PROC HomeSetup()
 !***********************************************************************
 !* Prozedur zum Programmieren und Parametrieren der Homepositionen 1-5 *
 !*     Procedure for programming and setup the home positions 1-5      *
 !***********************************************************************
 ! Gewaehlte Homeposition / Selected home position
 VAR num n_HomeSelect;
 ! richtigstellen der Homereihenfolge falls erste home deaktiviert / Set default home configuration
 IF b_HomeInUse{1}=FALSE b_HomeInUse:=[TRUE,FALSE,FALSE,FALSE,FALSE];
 WHILE TRUE DO
  TPErase;
  rerun1:
	! Home Liste wird Initialisiert / Create list of homes
  FOR i FROM 1 TO 5 DO
		IF b_HomeInUse{i} THEN
			listHome{i}.text:=listHomeConst{i}.text+st_Home_label{i};
		ELSE
			listHome{i}.text:="";
		ENDIF
  ENDFOR
  !
  ! Waehle Home Nummer
  st_UiHeader:=["Setup Home.","Setup Home, Waehle eine Homepos aus.","???"];
  st_UiMsgButtons3:=["Please select the Home you want to change.","Anzahl der Home aendern","???"];
  st_UiMsgButtons4:=["OK","Ok","???"];
  st_UiMsgButtons5:=["Finished","Beenden","???"];
  st_UiMsgButtons:=["","",st_UiMsgButtons3{n_Sp},st_UiMsgButtons4{n_Sp},st_UiMsgButtons5{n_Sp}];
	n_HomeSelect := UIListView(\Result:=br_UiAnswer\Header:=st_UiHeader{n_Sp},listHome
 	  \BtnArray:=st_UiMsgButtons\Icon:=iconInfo\DefaultIndex:=1);
  IF br_UiAnswer = 5 THEN
  	TPErase;
  	TPShow TP_LATEST;
    RETURN;
  ENDIF
  IF br_UiAnswer = 3 THEN
		! Anzahl der verwendeten Homes\Number of used homes
		st_UiHeader:=["Enter number of homes used","Anzahl der verwendeten Home Positonen","???"];
		st_UiMsgLine1:=["   count 1-5","   Anzahl 1-5","???"];
		n_Temp := UINumEntry(\Header:=st_UiHeader{n_Sp}\Message:=st_UiMsgLine1{n_Sp}\Icon:=iconInfo
			\InitValue:=1\MinValue:=1\MaxValue:=5\AsInteger);
		!
		TEST n_Temp
			CASE 1:
				b_HomeInUse:=[TRUE,FALSE,FALSE,FALSE,FALSE];
				b_HomeAkt:=[TRUE,FALSE,FALSE,FALSE,FALSE];
			CASE 2:
				b_HomeInUse:=[TRUE,TRUE,FALSE,FALSE,FALSE];
				b_HomeAkt:=[TRUE,TRUE,FALSE,FALSE,FALSE];
			CASE 3:
				b_HomeInUse:=[TRUE,TRUE,TRUE,FALSE,FALSE];
				b_HomeAkt:=[TRUE,TRUE,TRUE,FALSE,FALSE];
			CASE 4:
				b_HomeInUse:=[TRUE,TRUE,TRUE,TRUE,FALSE];
				b_HomeAkt:=[TRUE,TRUE,TRUE,TRUE,FALSE];
      CASE 5:
      	b_HomeInUse:=[TRUE,TRUE,TRUE,TRUE,TRUE];
      	b_HomeAkt:=[TRUE,TRUE,TRUE,TRUE,TRUE];
     ENDTEST
     GOTO rerun1;
	ENDIF
  !
  rerun2:
  ! was soll geaendert werden / what should be changed
  n_Temp :=0;
  st_UiHeader:=["Setup homepos edit Home_","Setup Home, bearbeite Home_","???"];
  st_UiMsgLine1:=["Modify the position Home_","aendere die Position der Home_","???"];
  st_UiMsgLine2:=["Modify the description for Home_","aendere die Beschreibung fuer die Home_","???"];
  st_UiMsgLine3:=["Activate the output for Home_","Aktiviere den Ausgang fuer die Home_","???"];
  st_UiMsgButtons3:=["Return","Zurueck","???"];
  st_UiMsgButtons4:=["OK","OK","???"];
  st_UiMsgButtons5:=["Finished","Beenden","???"];
  st_UiMsgButtons:=["","",st_UiMsgButtons3{n_Sp},st_UiMsgButtons4{n_Sp},st_UiMsgButtons5{n_Sp}];
  li_UiMsgList:=[["",st_UiMsgLine1{n_Sp}+NumToStr(n_HomeSelect,0)],["",st_UiMsgLine2{n_Sp}+NumToStr(n_HomeSelect,0)]
  	,["",st_UiMsgLine3{n_Sp}+NumToStr(n_HomeSelect,0)],["",""],["",""]];
  n_Temp := UIListView(\Result:=br_UiAnswer\Header:=st_UiHeader{n_Sp}+NumToStr(n_HomeSelect,0),li_UiMsgList
  		\BtnArray:=st_UiMsgButtons\Icon:=iconInfo\DefaultIndex:=1);
	IF br_UiAnswer = 5 THEN
		TPErase;
		TPShow TP_LATEST;
		RETURN;
	ENDIF
	! zurueck zur auswahl / back to selection
	IF br_UiAnswer=3 GOTO rerun1;
	! auswahl aendere Pos / Select home to change
	IF n_Temp=1 THEN
		br_UiAnswer:=0;
		st_UiHeader:=["Setup homepos edit Home_","Setup Home, neue Pos fuer Home_","???"];
		st_UiMsgLine1:=["Make the current Position the new Home_"+NumToStr(n_HomeSelect,0)+" positon!","Die aktuell Position wird als Home_"+NumToStr(n_HomeSelect,0)+" gespeichert!","???"];
		st_UiMsgButtons3:=["Return","Zurueck","???"];
		st_UiMsgButtons4:=["   Save    Position?","Position speichern!","???"];
		st_UiMsgButtons5:=["Finished","Beenden","???"];
		st_UiMsgButtons:=["","",st_UiMsgButtons3{n_Sp},st_UiMsgButtons4{n_Sp},st_UiMsgButtons5{n_Sp}];
		br_UiAnswer:= UIMessageBox (\Header:=st_UiHeader{n_Sp}+NumToStr(n_HomeSelect,0)
			\Message:=st_UiMsgLine1{n_Sp}\BtnArray:=st_UiMsgButtons\Icon:=iconWarning);
		IF br_UiAnswer = 5 THEN
			TPErase;
			TPShow TP_LATEST;
			RETURN;
		ENDIF
		! Pos fuer die jeweilige Home zuweisen / Pos assign for each Home
		IF br_UiAnswer = 4 THEN
			t_Home := CTool();
			t_home.robhold:=TRUE;
		TEST n_HomeSelect
			CASE 1:
				jpHome1 := CJointT();
				robjOHome1:=jpHome1.robax;
				extjOHome1:=jpHome1.extax;
			CASE 2:
				jpHome2 := CJointT();
				robjOHome2:=jpHome2.robax;
				extjOHome2:=jpHome2.extax;
			CASE 3:
				jpHome3 := CJointT();
				robjOHome3:=jpHome3.robax;
				extjOHome3:=jpHome3.extax;
			CASE 4:
				jpHome4 := CJointT();
				robjOHome4:=jpHome4.robax;
				extjOHome4:=jpHome4.extax;
			CASE 5:
				jpHome5 := CJointT();
				robjOHome5:=jpHome5.robax;
				extjOHome5:=jpHome5.extax;
			ENDTEST
			! ungueltig setzen / error set
			b_HomeAkt{n_HomeSelect}:=FALSE;
		GOTO rerun2;
	ENDIF
 ENDIF
 ! ruecksprung ins aenderungsmenue / jump back into the change of menu
 IF br_UiAnswer = 3 GOTO rerun2;
 ! auswahl aendere beschreibung / selection change description
 IF n_Temp=2 THEN
 	st_UiHeader:=["Setup homepos edit Home_","Setup Home, Beschreibung fuer Home_","???"];
	st_UiMsgLine1:=["Please enter the new description","Bitte eine Beschreibung fuer die HomePos eingeben.","???"];
	st_Home_label{n_HomeSelect} := UIAlphaEntry(\Header:=st_UiHeader{n_Sp}+NumToStr(n_HomeSelect,0),
	  \Message:=st_UiMsgLine1{n_Sp}\Icon:=iconInfo\InitString:= st_Home_label{n_HomeSelect});
	GOTO rerun2;
 ENDIF
 ! auswahl aktiviere Ausgang / Output enable selection
 IF n_Temp=3 THEN
	br_UiAnswer:=0;
	st_UiHeader:=["Setup homepos edit Home_","Setup Home, Ausgang fuer Home_","???"];
	st_UiMsgLine1:=["In order to activate the Home output, you must Warm Start the controller.","Der Ausgang fuer die Home wird durch einen Warmstart aktiviert!","???"];
	st_UiMsgButtons1:=["Warmstart!","Warmstart!","???"];
	st_UiMsgButtons3:=["Return","Zurueck","???"];
	st_UiMsgButtons5:=["Finished","Beenden","???"];
	st_UiMsgButtons:=[st_UiMsgButtons1{n_Sp},"",st_UiMsgButtons3{n_Sp},"",st_UiMsgButtons5{n_Sp}];
	br_UiAnswer:= UIMessageBox (\Header:=st_UiHeader{n_Sp}+NumToStr(n_HomeSelect,0)
	\Message:=st_UiMsgLine1{n_Sp}\BtnArray:=st_UiMsgButtons\Icon:=iconWarning);
	IF br_UiAnswer = 5 THEN
		TPErase;
		TPShow TP_LATEST;
		RETURN;
		ENDIF
		IF br_UiAnswer = 3 GOTO rerun2;
		IF br_UiAnswer = 1 WarmStart;
	ENDIF
 ENDWHILE
ENDPROC !(HomeSetup)

!*******************************************************************************

PROC SyncPosSetup()
 !******************************
 !*     Sync Switch Setup      *
 !******************************
 br_UiAnswer:=0;
 st_UiHeader:=["Setup SyncPos","Setup Synchron Position","???"];
 st_UiMsgLine1:=["Please note only use when the robot is at the ","Achtung  nur wenn der Roboter den Synchronschalter belegt","???"];
 st_UiMsgLine2:=["synchronous switch or on the soft-synchronous ","oder auf der Soft-Synchronposition steht","???"];
 st_UiMsgLine3:=["position. Otherwise, press> 'Abort'!","diese Position speichern. Ansonsten den Vorgang abbrechen!","???"];
 st_UiMsgButtons4:=["Save Position!","Position speichern!","???"];
 st_UiMsgButtons5:=["Abort","Abbruch","???"];
 st_UiMsgButtons:=["","","",st_UiMsgButtons4{n_Sp},st_UiMsgButtons5{n_Sp}];
 st_UiMsgLines:=[st_UiMsgLine1{n_Sp},st_UiMsgLine2{n_Sp},st_UiMsgLine3{n_Sp},"",""];
 br_UiAnswer:= UIMessageBox (\Header:=st_UiHeader{n_Sp}
		\MsgArray:=st_UiMsgLines\BtnArray:=st_UiMsgButtons\Icon:=iconWarning);
 IF br_UiAnswer = 5 THEN
	TPErase;
	TPShow TP_LATEST;
	RETURN;
 ENDIF
 ! Pos zuweisen
 IF br_UiAnswer = 4 THEN
	t_SMSync := CTool();
	t_SMSync.robhold:=TRUE;
	jpSM1SyncSwitch := CJointT(\TaskRef:=T_ROB1Id);
	robjOSM1SyncSwitch:=jpSM1SyncSwitch.robax;
	extjOSM1SyncSwitch:=jpSM1SyncSwitch.extax;
 ENDIF
 TPErase;
 TPShow TP_LATEST;
ENDPROC !(SynchPosSetup)

!*******************************************************************************

FUNC num n_RobInHomeDO()
 !*****************************************************************************************
 !* Funktion Ueberprueft die Home Ausgaenge des Roboters und gibt entsprechend 1-5 zurueck *
 !*        Function to return the number in which home the robot is at (1-5)              *
 !*****************************************************************************************
 !
 IF DOutput(SYS_do_Home_1)=1 THEN
   RETURN 1;
 ELSEIF DOutput(SYS_do_Home_2)=1 THEN
   RETURN 2;
 ELSEIF DOutput(SYS_do_Home_3)=1 THEN
   RETURN 3;
 ELSEIF DOutput(SYS_do_Home_4)=1 THEN
   RETURN 4;
 ELSEIF DOutput(SYS_do_Home_5)=1 THEN
   RETURN 5;
 ELSE
   RETURN 0;
 ENDIF
ENDFUNC !(n_RobInHomeDO)

!*******************************************************************************

FUNC bool b_PLCNeedHome(num n_H)
 !***********************************************************
 !* Function to check which home the PLC requires the robot *
 !***********************************************************
 !
 TEST n_H
 	CASE 1:
		IF DInput(PLC_di_Home_1)=1 RETURN TRUE;
 		RETURN FALSE;
  CASE 2:
 		IF DInput(PLC_di_Home_2)=1 RETURN TRUE;
  	RETURN FALSE;
  CASE 3:
  	IF DInput(PLC_di_Home_3)=1 RETURN TRUE;
  	RETURN FALSE;
  CASE 4:
  	IF DInput(PLC_di_Home_4)=1 RETURN TRUE;
  	RETURN FALSE;
  CASE 5:
  	IF DInput(PLC_di_Home_5)=1 RETURN TRUE;
  	RETURN FALSE;
  DEFAULT :
    	RETURN FALSE;
 ENDTEST
ENDFUNC !(b_PLCNeedHome)

!*******************************************************************************

PROC CheckValue(num Value,num MinValue,num MaxValue,num Dec,string Header)
 !**************************************************************************************************
 !*            Prozedur Ueberprueft ob ein Wert innerhalb eines Bereiches liegt                    *
 !* uebergebene Parameter: num Value,num MinValue,num MaxValue,num Dec,string Header (fuer meldung) *
 !*                         Check values are within certain paramaters                             *
 !**************************************************************************************************
 WHILE Value<MinValue OR Value>MaxValue DO
  st_UiHeader:=["Value Error ","Falscher Wert von ","???"];
  st_UiMsgLine1:=["The value is outside the Min or Max range.","Wert ist ausserhalb des gueltigen Bereichs","???"];
  st_UiMsgLine2:=["Min Value= ","Minnimal Wert= ","???"];
  st_UiMsgLine3:=["Max Value= ","Maximal  Wert= ","???"];
  st_UiMsgLine4:=["The Programmed Value=","Programmierter Wert= ","???"];
  UIMsgBox\Header:=st_UiHeader{n_Sp}+Header, st_UiMsgLine1{n_Sp}\MsgLine2:=st_UiMsgLine2{n_Sp}+NumToStr(MinValue,Dec)
 		 \MsgLine3:=st_UiMsgLine3{n_Sp}+NumToStr(MaxValue,Dec) \MsgLine4:=st_UiMsgLine4{n_Sp}+NumToStr(Value,Dec)
  		\Buttons:=btnOK\Icon:=iconWarning;
	Stop ;
	ENDWHILE
ENDPROC !(CheckValue)

!*******************************************************************************

PROC PowerOnCom()
 !***************************************************
 !* Abfrage der Appl im System nach einem Warmstart *
 !*        Check system after a warm start          *
 !***************************************************
 !Appl-Feld wird geloescht / Applications-deleted box
 VAR bool b_ComDummy:=FALSE;
 VAR bool b_timeout;
 VAR num n_ComDummy:=0;
 VAR NUM n_error_offset_x:=0 ;
 VAR NUM n_error_offset_y:=0 ;
 VAR NUM n_error_offset_z:=0 ;
 VAR bool b_ABS_Acc_Enable_MEM:=TRUE;
 VAR string st_CFG_RobotType;

 b_PwOnEnd:=FALSE;
 Reset VB_do_TaskBrake;
 FOR I FROM 1 TO 30 DO
	b_Start_present{I}:=TRUE;
	b_ReStart_present{I}:=TRUE;
	b_Stop_present{I}:=TRUE;
	b_Reset_present{I}:=TRUE;
 ENDFOR
 b_StartUser_present:=TRUE;
 b_ReStartUser_present:=TRUE;
 b_StopUser_present:=TRUE;
 b_ResetUser_present:=TRUE;
 ! Appl Info loeschen
 n_ApplMax:=0;
 n_Fk4ApplAktiv:=0;
 b_ABS_Acc_Enable:=TRUE;

 !Abfrage der einzelnen Appls / Check individual Applications
 n_ComDummy:=0;
 FOR I FROM 1 TO 30 DO
  b_ComDummy:=TRUE;
  st_Appl_Info{I,1}:="";
  st_Appl_Info{I,2}:="";
  st_Appl_Info{I,3}:="";
  ! aufruf der PowerOn jeder Appl und einlesen der Strings / calling the PowerOn Appl and read each of the strings
  n_Fk4ApplNum:=I;
  %"PowerON"+NumToStr(I,0)%;
  !
  IF b_ComDummy=TRUE THEN
    Incr n_ComDummy;
    st_Appl_Info{n_ComDummy,1}:=ValToStr(I);
    st_Appl_Info{n_ComDummy,2}:=st_Appl_Name;
    st_Appl_Info{n_ComDummy,3}:=st_Appl_Key{n_Sp};
 	  Incr n_ApplMax;
  ENDIF
 ENDFOR
 n_Fk4ApplNum:=0;

b_TbCom_Started:=FALSE ;

Waituntil b_TbCom_Started=TRUE\MaxTime:= 50\TimeFlag:= b_timeout;
!***************************
!* Waiting TB_Com to start *
!***************************

 b_PowerOn_exe_OK:=TRUE ;

 ! setzen der Homepos als Weltzonen / share of the world as Homepos Zones
 !
 IF b_HomeInUse{1}=TRUE THEN
    WZHomeJointDef \Inside, sh_HomePos1, jpHome1, delta_HomePosFine;
    WZDOSet \Stat,wz_HomePos1 \Inside, sh_HomePos1, SYS_do_Home_1,high;
    b_HomeAkt{1}:=TRUE;
 ENDIF
 !
 IF b_HomeInUse{2}=TRUE THEN
     WZHomeJointDef \Inside, sh_HomePos2, jpHome2, delta_HomePosFine;
     WZDOSet \Stat,wz_HomePos2 \Inside, sh_HomePos2, SYS_do_Home_2,high;
     b_HomeAkt{2}:=TRUE;
 ENDIF
 !
 IF b_HomeInUse{3}=TRUE THEN
     WZHomeJointDef \Inside, sh_HomePos3, jpHome3, delta_HomePosFine;
     WZDOSet \Stat,wz_HomePos3 \Inside, sh_HomePos3, SYS_do_Home_3,high;
     b_HomeAkt{3}:=TRUE;
 ENDIF
 !
 IF b_HomeInUse{4}=TRUE THEN
     WZHomeJointDef \Inside, sh_HomePos4, jpHome4, delta_HomePosFine;
     WZDOSet \Stat,wz_HomePos4 \Inside, sh_HomePos4, SYS_do_Home_4,high;
     b_HomeAkt{4}:=TRUE;
 ENDIF
 !
 IF b_HomeInUse{5}=TRUE THEN
     WZHomeJointDef \Inside, sh_HomePos5, jpHome5, delta_HomePosFine;
     WZDOSet \Stat,wz_HomePos5 \Inside, sh_HomePos5, SYS_do_Home_5,high;
     b_HomeAkt{5}:=TRUE;
 ENDIF
 !
 ! Poweron fuer Anwender wenn noetig / Poweron for users if necessary
 %"PowerOnUser"%;
 !---------------
 ! Copy SM_Files and Backup files
 SM1_CopyCfg;
 CopyCfg;

b_PwOnEnd:=TRUE;
b_ABS_Acc_Enable_MEM:=b_ABS_Acc_Enable;

 !Get robot type
 ReadCfgData "/MOC/ROBOT/ROB_1","use_robot_type",st_CFG_RobotType;

 st_RobotType:=st_CFG_RobotType;

 !Set Absoulute accuracy flag
 TEST st_RobotType

 CASE "ROB1_6620LX_1.90_150":
 	b_Robot_ABS_Type:=FALSE;
 DEFAULT:
 	b_Robot_ABS_Type:=b_ABS_Acc_Enable_MEM;
 ENDTEST

 !Set output as this robot does not use this output
 IF st_RobotType="ROB1_6620LX_1.90_150" Set SM1_do_Stopped;

 IF b_Robot_ABS_Type THEN
	! Abfrage ob die AbsAcc ein ist
	ReadCfgData "/MOC/ROBOT/ROB_1","use_robot_calib",st_Abs;

	IF st_Abs="r1_uncalib" THEN
		st_UiHeader:=["Com, Absolute Accuracy error","Com, Keine Absolutgenauigkeit","???"];
		st_UiMsgLine1:=["Warning!! The robot absolute accuracy is turned Off.","Ohne Absolutgenauigkeit ist es nicht erlaubt den Roboter ","???"];
		st_UiMsgLine2:=["There is a risk of collisions!","zu bewegen, es besteht Kollisionsgefahr!","???"];
		st_UiMsgLine3:=["Please ensure it is enabled!","Bitte schalten Sie die Absolutgenauigkeit wieder ein!","???"];
		ErrWrite st_UiHeader{n_Sp},st_UiMsgLine1{n_Sp} \RL2:=st_UiMsgLine2{n_Sp}\RL3:=st_UiMsgLine3{n_Sp};
	ELSE
		!Check absolute accurate data exist
		ReadCfgData "/MOC/ARM_CALIB/rob1_1", "error_offset_x", n_error_offset_x;
		ReadCfgData "/MOC/ARM_CALIB/Rob1_1", "error_offset_y", n_error_offset_y;
		ReadCfgData "/MOC/ARM_CALIB/Rob1_1","error_offset_z",n_error_offset_z;

		IF n_error_offset_x=0 AND n_error_offset_y=0 AND n_error_offset_z=0 THEN
			st_UiHeader:=["Com, Absolute Accuracy error","Com, Keine Absolutgenauigkeit","???"];
			st_UiMsgLine1:=["Warning!! The robot absolute accuracy is turned On but,","Warnung!! Der Roboter absolute Genauigkeit ist eingeschaltet,","???"];
			st_UiMsgLine2:=["the 'ARM/JOINT_CALIB' data in the 'MOC.cfg' file","aber die 'ARM/JOINT_CALIB' Daten in der 'MOC.cfg'","???"];
			st_UiMsgLine3:=["may not exist.","Datei kann nicht vorhanden","???"];
			st_UiMsgLine4:=["Please check.","Bitte überprüfen.","???"];

			ErrWrite st_UiHeader{n_sp},st_UiMsgLine1{n_sp} \RL2:=st_UiMsgLine2{n_sp}\RL3:=st_UiMsgLine3{n_sp}\RL4:=st_UiMsgLine4{n_sp};
		ENDIF
	ENDIF
 ENDIF

 ERROR
 !** Error Handler**
 SkipWarn;

 TEST ERRNO
 CASE ERR_CFG_NOTFND:
   TRYNEXT;

 CASE ERR_REFUNKPRC:
   b_ComDummy:=FALSE;
   st_Appl_Name:="";
   st_Appl_Key:=["","",""];
   TRYNEXT;
 ENDTEST
ENDPROC !(PowerOnCom)

!*******************************************************************************

PROC StartCom()
 !****************************
 !* Aufruf der Startroutinen *
 !*     Start Routine        *
 !****************************
 VAR bool b_ComDummy:=FALSE;
 VAR num n_ComDummy:=0;
 ! ob Programmzeiger versetzt wurde / whether program pointer was moved
 IF PPMovedInManMode() ResetPPMoved;
 !
 IF b_CheckPP=FALSE THEN
	Reset SYS_do_MainStarted;
	! loeschen von Fehlern wenn neustart / Clear errors after new start
	SetGO PLC_go_ErrCode, 0;
	Reset PLC_do_MsgToPLC;
	Reset PLC_do_ErrorToPLC;
	Reset PLC_do_StopToPLC;
	MsgBox_Clear;
	b_CollClearAct:= FALSE;
	n_JobReqNum:=0;
	n_JobFinNum:=0;
	b_JobF_w:=FALSE;
	b_JobR_w:=FALSE;
 ENDIF

 ! aufruf der Eventroutinen der Appl / calling the routines in the events
 b_UserEv:=FALSE;
 IF n_ApplMax >0 AND n_ApplMax< 31 THEN
	FOR I FROM 1 TO n_ApplMax DO
		n_Appl_count:=I;
		IF (st_Appl_Info{I,1}="") OR (b_Start_present{I}=FALSE) GOTO END_Start;
		b_ComDummy:=StrToVal(st_Appl_Info{I,1},n_ComDummy);
		%"Start"+NumToStr(n_ComDummy,0)%;
	 	END_Start:
	ENDFOR
 ENDIF

 IF n_ModeOP_Mem<>OpMode() THEN
      b_Ignore_NoAppl_Chk:=FALSE ;
      n_ModeOP_Mem:=OpMode();
 ENDIF

 IF PLC_di_NoApplication=1 AND b_Ignore_NoAppl_Chk=FALSE THEN
    MsgBoxEv_Clear;
    st_MsgBoxEvHeader:=["Warning!! StartCom","Warnung!! StartCom","???"];
	st_Dummy:=["You are about to run with (PLC_di_NoApplication=1)","Du bist zum Laufen (PLC_di_NoApplication=1)","???"];
	st_MsgBoxEvLine3:=["no Application selected.","nein Anwendung ausgewaehlt.","???"];
    st_MsgBoxEvbutton4:=["Continue","OK","???"];

	IF OpMode()<>OP_Auto THEN
		st_MsgBoxEvLine5:=["Press>'Ignore' to stop message re-occuring.","Druecke> 'Ignorieren' um die Nachricht zu stoppen.","???"];
		st_MsgBoxEvbutton5:=["Ignore","Ignorieren","???"];
   ENDIF

    MsgBoxEv\line1:=""\Line2:=st_Dummy{n_Sp};

    IF n_MsgBoxEvAnswer=5 b_Ignore_NoAppl_Chk:=TRUE;
 ENDIF

 b_UserEv:=TRUE;
 IF b_StartUser_present = TRUE %"StartUser"%;
 !
 ERROR
 !** Error Handler**
 IF ERRNO=ERR_REFUNKPRC THEN
 	SkipWarn;
	IF b_UserEv=TRUE THEN
		b_StartUser_present:=FALSE;
	ELSE
		b_Start_present{n_Appl_count}:=FALSE;
 	ENDIF
	TRYNEXT;
 ENDIF
ENDPROC !(StartCom)

!*******************************************************************************

PROC StopCom()
 !***************************
 !* Aufruf der Stoproutinen *
 !*     Stop Routine        *
 !***************************
 VAR bool b_ComDummy:=FALSE;
 VAR num n_ComDummy:=0;
 ! ob Programmzeiger versetzt wurde / whether program pointer was moved
 IF b_CheckPP=FALSE   Reset SYS_do_MainStarted;
 ! aufruf der Eventroutinen der Appl / calling the routines in the events
 b_UserEv:=FALSE;
 IF n_ApplMax >0 AND n_ApplMax< 31 THEN
	FOR I FROM 1 TO n_ApplMax DO
		n_Appl_count:=I;
		IF (st_Appl_Info{I,1}="") OR (b_Stop_present{I}=FALSE) GOTO END_Stop;
		b_ComDummy:=StrToVal(st_Appl_Info{I,1},n_ComDummy);
		%"Stop"+NumToStr(n_ComDummy,0)%;
	 	END_Stop:
	 ENDFOR
 ENDIF
 b_UserEv:=TRUE;
 IF b_StopUser_present = TRUE %"StopUser"%;
 ERROR
 !** Error Handler**
 IF ERRNO=ERR_REFUNKPRC THEN
 	SkipWarn;
	IF b_UserEv=TRUE THEN
		b_StopUser_present:=FALSE;
	ELSE
		b_Stop_present{n_Appl_count}:=FALSE;
 	ENDIF
	TRYNEXT;
 ENDIF
ENDPROC !(StopCom)

!*******************************************************************************

PROC RestartCom()
 !******************************
 !* Aufruf der ReStartroutinen *
 !*     Re-Start Routine       *
 !******************************
 VAR bool b_ComDummy:=FALSE;
 VAR num n_ComDummy:=0;
 VAR errnum errno1;
 ! ob Programmzeiger versetzt wurde / whether program pointer was moved
 b_PPMoved:=FALSE;
 IF PPMovedInManMode() THEN
	b_PPMoved:=TRUE;
	! loeschen von Fehlern wenn start / Clear errors if Restart
	SetGO PLC_go_ErrCode, 0;
	Reset PLC_do_MsgToPLC;
	Reset PLC_do_ErrorToPLC;
	Reset PLC_do_StopToPLC;
	MsgBox_Clear;
	MsgBoxEv_Clear;
	b_CollClearAct:= FALSE;
	b_JobF_w:=FALSE;
	b_JobR_w:=FALSE;

     IF DOutput(SYS_do_MainStarted)=1 AND DOutput (SYS_do_ApplRun)=1 AND b_PPMoved_mem=FALSE THEN
         b_PPMoved_mem:=TRUE;
         Log_Message "STD","Program pointer moved in Manual mode";
     ENDIF

 ENDIF

 IF OpMode()=OP_AUTO b_PPMoved_mem:=FALSE;

 IF b_CheckPP=FALSE   Reset SYS_do_MainStarted;
 ! aufruf der Eventroutinen der Appl / calling the routines in the events
 b_UserEv:=FALSE;
 IF n_ApplMax >0 AND n_ApplMax< 31 THEN
		FOR I FROM 1 TO n_ApplMax DO
			n_Appl_count:=I;
			IF (st_Appl_Info{I,1}="") OR (b_ReStart_present{I}=FALSE)  GOTO END_Restart;
			b_ComDummy:=StrToVal(st_Appl_Info{I,1},n_ComDummy);
			%"Restart"+NumToStr(n_ComDummy,0)%;
			END_Restart:
		ENDFOR
	ENDIF

 b_UserEv:=TRUE;
 IF b_ReStartUser_present = TRUE %"RestartUser"%;
 ! abfrage auf simulierte signale
 IF DOutput(VB_do_Simulated_IO)= 1 AND OpMode()= OP_AUTO  AND RobOs() = TRUE THEN
	! Meldung an SPS
	SetGO PLC_go_ErrCode, 34;
	Set PLC_do_MsgToPLC;
 	WHILE DOutput(VB_do_Simulated_IO)= 1 AND OpMode()= OP_AUTO DO
  		st_UiHeader:=["Com, Caution simulated signals!","Com, Achtung Simulierte Signale!","???"];
  		st_UiMsgLine1:=["There are some signals that are simulated which is not allowed in","Das Simulieren von Signalen ist im Automatik nicht erlaubt!","???"];
  		st_UiMsgLine2:=["automatic mode!  Please switch to manual mode,","In die Betriebsart Hand wechseln und die","???"];
  		st_UiMsgLine3:=["select the I/O menu then turn off the simulation/s.","Simulation aller Signale im Ein-Ausgangs Fenster ausschalten.","???"];
  		UIMsgBox\Header:=st_UiHeader{n_Sp},st_UiMsgLine1{n_Sp}\MsgLine2:=st_UiMsgLine2{n_Sp}\MsgLine3:=st_UiMsgLine3{n_Sp}
  						\Buttons:=btnNone\Icon:=iconError\MaxTime:=1.5\BreakFlag:=errno1;
			!
	ENDWHILE
 	SetGO PLC_go_ErrCode, 0;
 	Reset PLC_do_MsgToPLC;
 ENDIF
 ! check SafeMove function,at error to reduce speed
 IF DOutput(SM1_do_BrakeReq) =0 THEN
  	VelSet 100,5000;
 ELSE
  	VelSet 100,150;
		ErrWrite \W, "ComBase, SM1_do_BrakeReq =1", "Speed reduce to 150mm/s" ;
 ENDIF

 IF n_ModeOP_Mem<>OpMode() THEN
      b_Ignore_NoAppl_Chk:=FALSE ;
      n_ModeOP_Mem:=OpMode();
 ENDIF

ResetPPMoved;

 ERROR
 !** Error Handler**
 IF ERRNO=ERR_REFUNKPRC THEN
 	SkipWarn;
	IF b_UserEv=TRUE THEN
		b_ReStartUser_present:=FALSE;
	ELSE
		b_ReStart_present{n_Appl_count}:=FALSE;
 	ENDIF
	TRYNEXT;
 ENDIF
ENDPROC !(RestartCom)

!*******************************************************************************

PROC ResetCom()
 !****************************
 !* Aufruf der Resetroutinen *
 !*      Reset Routine       *
 !****************************
 VAR bool b_ComDummy:=FALSE;
 VAR num n_ComDummy:=0;
 ! aufruf der Eventroutinen der Appl / calling the routines in the events
 b_UserEv:=FALSE;
 IF n_ApplMax >0 AND n_ApplMax< 31 THEN
	FOR I FROM 1 TO n_ApplMax DO
		n_Appl_count:=I;
		IF (st_Appl_Info{I,1}="") OR (b_Reset_present{I}=FALSE) GOTO END_Reset;
		b_ComDummy:=StrToVal(st_Appl_Info{I,1},n_ComDummy);
		%"Reset"+NumToStr(n_ComDummy,0)%;
	 	END_Reset:
	ENDFOR
 ENDIF
 b_UserEv:=TRUE;
 IF b_ResetUser_present = TRUE %"ResetUser"%;
 ERROR
 !** Error Handler**
 IF ERRNO=ERR_REFUNKPRC THEN
 	SkipWarn;
	IF b_UserEv=TRUE THEN
		b_ResetUser_present:=FALSE;
	ELSE
		b_Reset_present{n_Appl_count}:=FALSE;
 	ENDIF
	TRYNEXT;
 ENDIF
ENDPROC !(ResetCom)

!*******************************************************************************

FUNC bool b_RobInHomeDO(num Home)
 !************************************************************************************
 !*                            Funktion b_RobInHomeDO                                *
 !* Funktion Ueberprueft die Home Ausgaenge des Roboters und gibt FALSE/TRUE zurueck *
 !*     Function checks the robot exits the home and gives FALSE / TRUE back         *
 !************************************************************************************
  IF Home = 1 AND DOutput(SYS_do_Home_1)=1 THEN
    RETURN TRUE;
  ELSEIF Home = 2 AND DOutput(SYS_do_Home_2)=1 THEN
    RETURN TRUE;
  ELSEIF Home = 3 AND DOutput(SYS_do_Home_3)=1 THEN
    RETURN TRUE;
  ELSEIF Home = 4 AND DOutput(SYS_do_Home_4)=1 THEN
    RETURN TRUE;
  ELSEIF Home = 5 AND DOutput(SYS_do_Home_5)=1 THEN
    RETURN TRUE;
  ELSE
    RETURN FALSE;
  ENDIF
ENDFUNC !(b_RobInHomeDO)

!*******************************************************************************

PROC SM1_CopyCfg()
 !**********************************************
 !* Routine to copy savemove config cfg files  *
 !**********************************************

 VAR string stSMCalFileInt;
 VAR string stSMFileInt;
 VAR string stSMCalFileHome;
 VAR string stSMFileHome;
 VAR string stSMCalFileBck;
 VAR string stSMFileBck;
 VAR string stBckName;
 VAR num n_index;
 ! create folder
 MakeDir "HOME:/SafetyBCK";
 FOR i FROM 1 TO 4 DO
 	! Check all files
	stSMCalFileHome:= stSMCalHome+ ValToStr(i)+ ".xml";
  stSMCalFileInt:= stSMCalInternal+ ValToStr(i)+ ".xml";
  stSMFileHome:= stSMHome+ ValToStr(i)+ ".sxml";
  stSMFileInt:= stSMInternal+ ValToStr(i)+ ".sxml";
  ! If file has a config then safe to Home
	IF FileSize(stSMFileInt) > nSMFilesize THEN
	  	IF IsFile(stSMFileHome) THEN
	   		! delete existing file at Homefolder
	  		RemoveFile stSMFileHome;
	 	  ENDIF
	    IF IsFile(stSMCalFileHome) THEN
	   		! delete existing file at Homefolder
	  		RemoveFile stSMCalFileHome;
	    ENDIF
	    ! Copy actual config from System
	 		CopyFile stSMFileInt, stSMFileHome;
	 		CopyFile stSMCalFileInt, stSMCalFileHome;
			! Read Pin code
			WaitTime 0.2;
			IF IsFile(stSMFileHome) n_SMPins{i}:= GetPinCode(stSMFileHome);
	 ELSE
	 		! Read Backup name
			n_index:=0;
			ReadCfgData "/MMC/BACKUP_DEFAULT/backup_path//hd0a/BACKUP","backup_name",stBckName\ListNo:=n_index;
			stSMFileBck:= stSMBck+ stBckName+ stSMBckFile+ ValToStr(i)+ ".sxml";
			stSMCalFileBck:= stSMBck+ stBckName+ stSMBckCal+ ValToStr(i)+ ".xml";
			! Check on exist config at Backupfolder and right Pin
			! it is for restoring SafeMove config
			IF  IsFile(stSMFileBck)THEN
				 IF (n_SMPins{i} = GetPinCode(stSMFileBck)) THEN
		  			! delete existing file and Copy actual config to System
			  		RemoveFile stSMFileInt;
	  				CopyFile stSMFileBck, stSMFileInt;
		  			ErrWrite \I, "Com, PowerON", "SafeMove, Configfile re-established";
			  		IF  IsFile(stSMCalFileBck)THEN
			  			RemoveFile stSMCalFileInt;
				  		CopyFile stSMCalFileBck, stSMCalFileInt;
					  	ErrWrite \I, "Com, PowerON", "SafeMove, Calfile re-established";
					  ENDIF
			 	 ENDIF
			ENDIF
		ENDIF
 ENDFOR
 !
 ERROR
 !** Error Handler**
 IF ERRNO = ERR_FILEEXIST THEN
  	SkipWarn;
	!Do Nothing
 ELSEIF ERRNO = ERR_FILEACC THEN
  	SkipWarn;
	TRYNEXT;
 ENDIF
 IF ERRNO = ERR_CFG_NOTFND THEN
 	ErrWrite "ComBase /PowerOn", "Path to save SM-Data not correct!" \RL2:="Change the Path in SM1_CopyCfg";
 ENDIF
ENDPROC !(SM1_CopyCfg)

!*******************************************************************************

PROC CopyCfg()
 !************************************************
 !* Routine to copy config cfg files for backup  *
 !************************************************

 VAR string stBckName;
 VAR num n_index;

 ! create folder
 MakeDir "HOME:";

 !Get Backuip name
 ReadCfgData "/MMC/BACKUP_DEFAULT/backup_path//hd0a/BACKUP","backup_name",stBckName\ListNo:=n_index;

 !Create backup Directory name
  IF RobOS() THEN
     stCon_Int_Dir:="/hd0a/internal";
     stCon_Home_Dir:="/hd0a/"+stBckName+"/Home";
     sthd0a_Home_Dir:="/hd0a/Backup/"+stBckName+"/Home";
 ELSE
    stCon_Int_Dir:="INTERNAL:";
    stCon_Home_Dir:="HOME:";
    sthd0a_Home_Dir:="HOME:";
 ENDIF

 !Copy IPaddress file to internal home directory
 IF IsFile(stCon_Int_Dir + "/mc.cfg") THEN

   !Delete old file
    IF IsFile(stCon_Home_Dir + "/mc.cfg") RemoveFile stCon_Home_Dir + "/mc.cfg";

    CopyFile stCon_Int_Dir + "/mc.cfg",stCon_Home_Dir + "/mc.cfg";
 ELSEIF IsFile(sthd0a_Home_Dir + "/mc.cfg") THEN
    CopyFile sthd0a_Home_Dir + "/mc.cfg",stCon_Int_Dir + "/mc.cfg";
 ENDIF

 !Copy UAS files to internal home directory
 IF IsFile(stCon_Int_Dir + "/uas_groups.xml") THEN

   !Delete old file
    IF IsFile(stCon_Home_Dir + "/uas_groups.xml") RemoveFile stCon_Home_Dir + "/uas_groups.xml";

    CopyFile stCon_Int_Dir + "/uas_groups.xml",stCon_Home_Dir + "/uas_groups.xml";
 ELSEIF IsFile(sthd0a_Home_Dir + "/uas_groups.xml") THEN
    CopyFile sthd0a_Home_Dir + "/uas_groups.xml",stCon_Int_Dir + "/uas_groups.xml";
 ENDIF

  IF IsFile(stCon_Int_Dir + "/uas_users.xml") THEN

   !Delete old file
    IF IsFile(stCon_Home_Dir + "/uas_users.xml") RemoveFile stCon_Home_Dir + "/uas_users.xml";

    CopyFile stCon_Int_Dir + "/uas_users.xml",stCon_Home_Dir + "/uas_users.xml";
 ELSEIF IsFile(sthd0a_Home_Dir + "/uas_users.xml") THEN
    CopyFile sthd0a_Home_Dir + "/uas_users.xml",stCon_Int_Dir + "/uas_users.xml";
 ENDIF

 RETURN;

 ERROR
 !** Error Handler**

 TEST ERRNO
 CASE ERR_FILEEXIST:
  	SkipWarn;
	!Do Nothing
 CASE ERR_FILEACC:
  	SkipWarn;
	TRYNEXT;
 !Case ERR_CFG_NOTFND:
 !	ErrWrite "ComBase /PowerOn", "Path to save SM-Data not correct!" \RL2:="Change the Path in SM1_CopyCfg";
 ENDTEST

ENDPROC !(SM1_CopyCfg)

!*******************************************************************************

PROC SM1_SyncMove()
 !*******************************
 !* Check Save Move Sync Switch *
 !*******************************
 !
 MoveAbsJ jpSM1SyncSwitch, v500, fine, t_SMSync;
 WaitTime \InPos, 1;
 n_Step:=1;
 WaitDI SM1_di_SyncSwitch ,1\MaxTime:=3;
 !*******************************
 !* Waiting for SyncSwith Input *
 !*******************************

 n_Step:=2;
 WaitDO SM1_do_Synced ,1\MaxTime:=3;
 !*******************************
 !*    Waiting for Sync Ouput   *
 !*******************************

 IF DOutput(SM1_do_Synced) =1 THEN
	VelSet 100,5000;
 ELSE
	VelSet 100,150;
 ENDIF
 ERROR
 SkipWarn;
 !** Error Handler**
 IF ERRNO=ERR_WAIT_MAXTIME THEN
  TEST n_Step
   	CASE 1:
			st_MsgBoxHeader:=["Waiting for Syncronisation Switch signal","Warte auf den Synchronschalter","???"];
			st_MsgBoxLine3:=["Please check the Safemove Sync Switch","ueberpruefe den Synchronschalter","???"];
			st_MsgBoxLine4:=["Please check the robot position or calibration.","ueberpruefe die Roboterposition/Kalibrierung","???"];
			st_MsgBoxLine5:=["","","???"];
			st_MsgBoxbutton4:=["Retry","Wiederhole","???"];
			st_MsgBoxbutton5:=["Abort","Abbruch","???"];
			st_MsgBoxGeraeteName:=["SafeMove","SafeMove","???"];
			n_MsgBoxGeraeteNr:=1;
			st_MsgBoxSignal:="SM1_di_SyncSwitch";
			st_MsgBoxSignalValue:="1";
			n_MsgBoxApplError:=0;
			!Fehler Nummer an die SPS\Error Number to the PLC
			n_MsgBoxPLC_Error:=41;
			st_MsgBoxElogLine4:="ComBase/SM1_SyncMove";
			MsgBox \diBreakSignal:=SYS_di_ErrReset;
			!
			TEST n_MsgBoxAnswer
				CASE 0:
					RETRY;
				CASE 4:
					RETRY;
				CASE 5:
					TRYNEXT;
			ENDTEST
   	CASE 2:
			st_MsgBoxHeader:=["Waiting for Safe Move Synchronised","Warte auf SafeMove Synchronisiert","???"];
			st_MsgBoxLine3:=["Please check the safe move configuration","ueberpruefe SafeMove konfiguration","???"];
			st_MsgBoxLine4:=["but, this is not possible in Automatic mode.","Automatikbetrieb ist bis zur Fehlerbehebung nicht moeglich","???"];
			st_MsgBoxLine5:=["","","???"];
			st_MsgBoxbutton5:=["Abort","Abbruch","???"];
			st_MsgBoxGeraeteName:=["SafeMove","SafeMove","???"];
			n_MsgBoxGeraeteNr:=1;
			st_MsgBoxSignal:="SM1_do_Synced";
			st_MsgBoxSignalValue:="1";
			n_MsgBoxApplError:=0;
			!Fehler Nummer an die SPS
			n_MsgBoxPLC_Error:=42;
			st_MsgBoxElogLine4:="ComBase/SM1_SyncMove";
			MsgBox \diBreakSignal:=SYS_di_ErrReset;
			!
			TEST n_MsgBoxAnswer
				CASE 0:
					TRYNEXT;
				CASE 5:
					TRYNEXT;
			ENDTEST
			DEFAULT:
			ErrWrite "n_Step Case Err"," ";
			!n_SW_WO_Step Case Err";
			Stop;
  	ENDTEST
 ENDIF
ENDPROC !(SM1_SyncMove)

!*******************************************************************************

PROC BrakeTest_CTRL()
 !*******************************
 !* Brake check control routine *
 !*******************************

 VAR num n_HomeMem;
 VAR signaldo alias_do;
 VAR string sTemp;
 VAR num n_FirstHome:=0;
 VAR jointtarget jpCurrentPos;

 WaitRob \InPos;

 !Determine which home the robot is at
 FOR i From 1 TO 5 DO
      sTemp:="SYS_do_Home_" + NumToStr(i,0);

      AliasIO sTemp, alias_do;

      IF DOutput(alias_do)=1 AND b_HomeAkt{i} AND n_FirstHome=0 THEN
          n_FirstHome:=i;
      ENDIF
 ENDFOR

 MsgBox_Clear;

 !Check if the robot is in a home
 IF n_FirstHome=0 THEN

     IF OpMode()=OP_AUTO THEN
         WHILE TRUE DO
            st_MsgBoxHeader:=["ComBase, Brake Test","ComBase, Bremsentest","???"];
            st_Dummy:=["Brake test operation in Automatic mode","Bremsentest in Automatikmodus","???"];
            st_Dummy2:=["but, the robot is not in any home position.","aber der Roboter ist nicht in einer Home-Position.","???"];

            st_MsgBoxLine4:=["Check why the robot is not in any home position.","Ueberpruefen warum Roboter nicht in einer Home-Pos ist","???"];
            st_MsgBoxLine5:=["Process cannot continue.","Prozess kann nicht weitergefuerht werden","???"];
            st_MsgBoxbutton5:=["OK","OK","???"];

            !Fehler Nummer an die SPS\Error number to the PLC
            n_MsgBoxPLC_Error:=109;
            st_MsgBoxElogLine4:="ComBase/BrakeTest_CTRL";
            MsgBox\Line1:=st_Dummy{n_Sp}\Line2:=st_Dummy2{n_Sp} \ErrorToPLC;

            Stop;
         ENDWHILE
     ELSE
        st_UiHeader:=["ComBase, Brake Test","ComBase Bremsentest, ","???"];
        st_UiMsgLine1:=["Brake test operation in Manual mode","Bremsentest in handmodus","???"];
        st_UiMsgLine2:=["but, the robot is not in any home position.","aber der Roboter ist nicht in einer Home-Position","???"];
        st_UiMsgLine5:=["Brake test will be carried out in the current position.","Bremsentest wird in der aktuellen Position ausgefuehrt","???"];
        st_UiMsgButtons5:=["OK","OK","???"];

		st_UiMsgButtons:=["","","","",st_UiMsgButtons5{n_Sp}];
		st_UiMsgLines:=[st_UiMsgLine1{n_Sp},st_UiMsgLine2{n_Sp},"","",st_UiMsgLine5{n_Sp}];

		br_UiAnswer:=UIMessageBox (\Header:=st_UiHeader{n_Sp}\MsgArray:=st_UiMsgLines\BtnArray:=st_UiMsgButtons \Icon:=iconError);

     	jpCurrentPos := CJointT();
        br_UiAnswer:=0;

		WHILE ABS(jpCurrentPos.extax.eax_a) <= 5 AND br_UiAnswer<>4 DO
		 	br_UiAnswer:=0;
			st_UiHeader:=["Com, Brake Test","Com, Bremsentest","???"];
			st_UiMsgLine1:=["Warning! The Linear track axis 7 is near 0mm and may fail braketest.","Achtung, die Achse 7 ist nahe 0 mm der Bremsentest koennte fehlschlagen","???"];

			st_UiMsgLine3:=["Select 'Ignore' to start the Brake Test at current position.","Mit 'ignorieren' wird der Bremsentest in der aktuellen Position gestartet.","???"];
			st_UiMsgLine4:=["Select 'Jog' then please move the axis >5 mm then 'Play' to start test.","Mit 'Jog' Bitte die Achse min. >5 mm. bewegen, mit 'Play' Test starten","???"];

            st_UiMsgButtons4:=["Ignore","ignorieren","???"];
			st_UiMsgButtons5:=["Jog","Jog","???"];

			st_UiMsgButtons:=["","","",st_UiMsgButtons4{n_Sp},st_UiMsgButtons5{n_Sp}];
			st_UiMsgLines:=[st_UiMsgLine1{n_Sp},"",st_UiMsgLine3{n_Sp},st_UiMsgLine4{n_Sp},""];

			br_UiAnswer:=UIMessageBox (\Header:=st_UiHeader{n_Sp}\MsgArray:=st_UiMsgLines\BtnArray:=st_UiMsgButtons \Icon:=iconError);

            IF br_UiAnswer=5 THEN
                ClearPath;
                Stop;
            ENDIF

            jpCurrentPos := CJointT();
        ENDWHILE
     ENDIF
 ENDIF

!Store current positional data
t_Home := CTool();
t_home.robhold:=TRUE;
jpCurrentPos:=CJointT();

!Call brake test routine
IF DOutput(SM1_do_BrakeOk) = 0 	VelSet 100, 150;

!Execute braketest call
SM1_BrakeTest;

!Ensure robot is back in correct position
 TEST n_FirstHome

    CASE 0:
        MoveAbsJ jpCurrentPos\NoEoffs, v1000, fine, t_Home;
    CASE 1:
        MoveAbsJ jpHome1\NoEoffs, v1000, fine, t_Home;
    CASE 2:
        MoveAbsJ jpHome2\NoEoffs, v1000, fine, t_Home;
    CASE 3:
        MoveAbsJ jpHome3\NoEoffs, v1000, fine, t_Home;
    CASE 4:
        MoveAbsJ jpHome4\NoEoffs, v1000, fine, t_Home;
    CASE 5:
        MoveAbsJ jpHome5\NoEoffs, v1000, fine, t_Home;
 ENDTEST

ENDPROC !(BrakeTest_CTRL)

!*******************************************************************************

PROC SM1_BrakeTest()
 !**********************************
 !* Check Save Move Brake Function *
 !**********************************
 VAR bool b_retryBrake;
 WaitTime \InPos, 1;
 ReRunBrake1:
 CyclicBrakeCheck_V2;

 WaitTime 0.2;
 IF (DOutput(SM1_do_BrakeReq) = 1)	THEN
 	st_MsgBoxHeader:=["ComBase, Wait for brake test OK","ComBase, Warte auf Bremsentest i.O.","???"];
	st_MsgBoxLine3:=["There was an problem during the brake test and the","Ueberpruefung der Bremse ist fehlgeschlagen!","???"];
        st_MsgBoxLine4:=["Brake test required signal from the controller is","Bremsentest Anforderung vom Controller steht an.","???"];
        st_MsgBoxLine5:=["still on. Please repeat the test again.","Bremsentest muss wiederholt werden.","???"];
	st_MsgBoxbutton5:=["Ok","Ok","???"];
	st_MsgBoxGeraeteName:=["SafeMove","SafeMove","???"];
	n_MsgBoxGeraeteNr:=1;
	st_MsgBoxSignal:="SM1_do_BrakeReq";
	st_MsgBoxSignalValue:="0";
	n_MsgBoxApplError:=0;
	!Fehler Nummer an die SPS\Error number to the PLC
	n_MsgBoxPLC_Error:=43;
	st_MsgBoxElogLine4:="ComBase/SM1_BrakeTest Request";
	MsgBox \diBreakSignal:=SYS_di_ErrReset;
	GOTO ReRunBrake1;
 ENDIF

 WaitUntil (DOutput(SM1_do_BrakeOk) = 1 OR  DOutput(SM1_do_BrakeLimit) = 1) AND DOutput(SM1_do_BrakeFault)= 0\MaxTime:=1;
 !*******************************************************
 !* Waiting for brake test to be satisfactory completed *
 !*******************************************************

 IF b_retryBrake=TRUE THEN
 	b_retryBrake:=FALSE;
	GOTO ReRunBrake1;
 ENDIF

 IF DOutput(SM1_do_BrakeOk) =1 OR DOutput(SM1_do_BrakeLimit) =1 THEN
  	VelSet 100,5000;
 ELSE
  	VelSet 100,150;
 ENDIF
 !
 ERROR
 !** Error Handler**

 MsgBox_Clear;

 SkipWarn;
 IF ERRNO=ERR_WAIT_MAXTIME THEN
	st_MsgBoxHeader:=["Wait for brake test OK","Warte auf SafeMove Bremsentest i.O.","???"];
	IF DOutput(SM1_do_BrakeFault) = 1 THEN
 		st_MsgBoxLine3:=["The robot motor brake/s are not","Die minimale Bremskraft ist nicht erreicht!","???"];
   		st_MsgBoxLine4:=["holding and must be replaced.","Defekte Bremse muss getauscht werden","???"];
 	ELSE
  		st_MsgBoxLine3:=["There was an problem during Robot motor","Ueberpruefung der Bremse war NIO","???"];
  		st_MsgBoxLine4:=["Brake test, please repeat test.","Bremsentest muss wiederholt werden","???"];
  	ENDIF
	st_MsgBoxLine5:=["With this fault, Automatic mode is not possible!!!","Automatikbetrieb ist bis zur Fehlerbehebung nicht moeglich","???"];
	st_MsgBoxbutton3:=["Retry","Wiederholen","???"];
	st_MsgBoxbutton5:=["Ok","Ok","???"];
	st_MsgBoxGeraeteName:=["SafeMove","SafeMove","???"];
	n_MsgBoxGeraeteNr:=1;
	st_MsgBoxSignal:="(BrakeOk OR BrakeWarn) AND BrakeNio=0";
	st_MsgBoxSignalValue:="";
	n_MsgBoxApplError:=0;

	!Fehler Nummer an die SPS\Error number to the PLC
	n_MsgBoxPLC_Error:=43;
	st_MsgBoxElogLine4:="ComBase/SM1_BrakeTest";
	MsgBox \diBreakSignal:=SYS_di_ErrReset;
	TEST n_MsgBoxAnswer
		CASE 0:
			TRYNEXT;
		CASE 3:
			b_retryBrake:=TRUE;
			TRYNEXT;
		CASE 5:
			TRYNEXT;
	ENDTEST
 ENDIF
ENDPROC !(SM1_BrakeTest)

!*******************************************************************************

PROC ManSyncService()
 !--------------------------------------------------------------
 ! function/Funktion: Procedure manuelle Synchronfahrt / manual SyncMove
 !
 ! state/Stand: 29.08.2011
 !
 ! author/Ersteller: Ramacher
 !--------------------------------------------------------------
 VAR jointtarget jpTempPos:=[ [ 0, 0, 0, 0, 0, 0],[0, 0, 0, 0, 0, 0]];
 VAR Bool b_ManSyncInt_Found:=TRUE;
 VAR Bool b_SetUpWasSelected:=FALSE;

 n_ManSyncCMD:=-2 ;
 !Test if 'ManSyncIntPos' routine exist
 %"ManSyncIntPos"%;
 n_ManSyncCMD:=-2 ;

 ReRun1:

 br_UiAnswer:=0;

 st_UiHeader:=["Com, CalibPos to move","Com, Kalibrierposition anfahren","???"];
 st_UiMsgLine1:=["Before the robot can be synchronised ensure it is","Bevor der Roboter synchronisiert werden kann, ist die","???"];
 st_UiMsgLine2:=["at the calibration position and the calib marks are","Kalibrierposition anzufahren und die Markierungen zu","???"];
 st_UiMsgLine3:=["          ***  Visuslly checked!  ***","      ***   KONTROLLIEREN !  ***","???"];
 st_UiMsgLine4:=["Where necessary, the calibration can be realised using","Mit Setup wird festgelegt ob die Markierungen mit einer oder zwei Positionen","???"];

 IF b_TwoSyncPos=FALSE THEN
 	st_UiMsgLine5:=["two separate positions. Current Setting = One position.","angefahren werden. Eingestellt:= Eine Position","???"];
 ELSE
 	st_UiMsgLine5:=["one position. Current Setting = Two seperate positions.","angefahren werden. Eingestellt:= Zwei Positionen","???"];
 ENDIF
 !
 st_UiMsgButtons1:=["Setup","Setup","???"];
 st_UiMsgButtons4:=["Move To","Anfahren","???"];
 st_UiMsgButtons5:=["Abort","Abbruch","???"];
 st_UiMsgButtons:=[st_UiMsgButtons1{n_Sp},"","",st_UiMsgButtons4{n_Sp},st_UiMsgButtons5{n_Sp}];
 st_UiMsgLines:=[st_UiMsgLine1{n_Sp},st_UiMsgLine2{n_Sp},st_UiMsgLine3{n_Sp},st_UiMsgLine4{n_Sp},st_UiMsgLine5{n_Sp}];
 !
 br_UiAnswer:=UIMessageBox (\Header:=st_UiHeader{n_Sp}\MsgArray:=st_UiMsgLines\BtnArray:=st_UiMsgButtons
							\Icon:=iconInfo);
TEST br_UiAnswer
	CASE 1: ! Setup
 		ReRun3:

        b_SetUpWasSelected:=TRUE;
 		br_UiAnswer:=0;
 		st_UiHeader:=["Com, Calib Pos-Setup","Com, Kalibrierpositions-Setup","???"];
 		st_UiMsgLine1:=["If the calibration position cannot be reached the with","Ist die Kalibrierposition nicht gleichzeitig mit allen ","???"];
 		st_UiMsgLine2:=["all axes at the same time, two positions can be used.","Achsen zu ereichen, koennen hier zwei Positionen gespeichert werden.","???"];
 		st_UiMsgLine4:=["The current setting is: ","Die aktuelle Einstellung ist: ","???"];

        IF b_TwoSyncPos=FALSE THEN
 			st_UiMsgLine5:=["One position.","Eine Position","???"];
 		ELSE
 			st_UiMsgLine5:=["Two seperate positions.","Zwei Positionen","???"];
 		ENDIF
 		!
 		IF b_TwoSyncPos=FALSE THEN
 			st_UiMsgButtons1:=["","",""];
 		ELSE
 			st_UiMsgButtons1:=["Set positions","Positionen festlegen","???"];
 		ENDIF

 		st_UiMsgButtons3:=["One Position ","Eine  Position_ ","???"];
 		st_UiMsgButtons4:=["Two Positions","Zwei Positionen","???"];
 		st_UiMsgButtons5:=["Back","Zurueck","???"];
 		st_UiMsgButtons:=[st_UiMsgButtons1{n_Sp},"",st_UiMsgButtons3{n_Sp},st_UiMsgButtons4{n_Sp},st_UiMsgButtons5{n_Sp}];
 		st_UiMsgLines:=[st_UiMsgLine1{n_Sp},st_UiMsgLine2{n_Sp},"",st_UiMsgLine4{n_Sp}+st_UiMsgLine5{n_Sp},""];
 		!
 		br_UiAnswer:=UIMessageBox (\Header:=st_UiHeader{n_Sp}\MsgArray:=st_UiMsgLines\BtnArray:=st_UiMsgButtons\Icon:=iconInfo);
 		TEST br_UiAnswer
 			CASE 1: ! Setup, Positionfestlegen
  			    ReRun2:

 				br_UiAnswer:=0;
 				st_UiHeader:=["Com, Calib Pos-Setup","Com, Kalibrierposition-Setup","???"];
 				st_UiMsgLine1:=["Please move the robot to the two positions","Bitte nacheinander den Roboter auf ein der beiden","???"];
 				st_UiMsgLine2:=["When you are sure the robot is at the correct","Positionen stellen, die Oberflaeche starten und mit den","???"];
 				st_UiMsgLine3:=["position, teach the positions.","Tasten die Positionen speichern. ","???"];
 				st_UiMsgLine4:=["Pos 1: Axis 1 to zero degrees. Axis 2-6 & external any other position.","Pos 1: Achse 1 fest auf 0 Grad, 2-6 u. ext. Achsen sind frei programmierbar","???"];
 				st_UiMsgLine5:=["Pos 2: Axis 2-6 & external to zero degrees, Axis 1 any other position.","Pos 2: Achsen 2-6 u. ext. Achse fest auf 0 Grad, 1 ist frei programmierbar","???"];
 				!
 				st_UiMsgButtons2:=["Teach Pos1","Pos 1 speichern","???"];
 				st_UiMsgButtons3:=["Teach Pos2","Pos 2 speichern","???"];
 				st_UiMsgButtons4:=["   SyncPos Teach/Info","Info SyncPos","???"];
 				st_UiMsgButtons5:=["Back","Zurueck","???"];
 				st_UiMsgButtons:=["",st_UiMsgButtons2{n_Sp},st_UiMsgButtons3{n_Sp},st_UiMsgButtons4{n_Sp},st_UiMsgButtons5{n_Sp}];
 				st_UiMsgLines:=[st_UiMsgLine1{n_Sp},st_UiMsgLine2{n_Sp},st_UiMsgLine3{n_Sp},st_UiMsgLine4{n_Sp},st_UiMsgLine5{n_Sp}];
 				!
 				br_UiAnswer:=UIMessageBox (\Header:=st_UiHeader{n_Sp}\MsgArray:=st_UiMsgLines\BtnArray:=st_UiMsgButtons	\Icon:=iconInfo);
 				IF br_UiAnswer=5 GOTO ReRun1;
 				IF br_UiAnswer=2 THEN
 					jpCalibPos1 := CJointT();
					jpCalibPos1.robax.rax_1 := 0;
 				ENDIF

 				IF br_UiAnswer=3 THEN
 					jpTemp := CJointT();
					jpCalibPos2:=jpCalibA1_A6;
					jpCalibPos2.robax.rax_1 := jpTemp.robax.rax_1;
 				ENDIF

				IF br_UiAnswer=4 THEN
					br_UiAnswer:=0;
 					st_UiHeader:=["Synchronisation Position Info","Info Synchron Position","???"];
 					st_UiMsgLine1:=["When using two separate positions for synchronisation, it is","Bei zwei Positionen fuer die Markierungstellung ist es","???"];
 					st_UiMsgLine2:=["recommended the second position is taught on the calibration marks.","sinnvoll die Synchronposition mit der 2. Position gleich zu setzen.","???"];
 					st_UiMsgLine3:=["If the robot is at Position 2, continue to save the position.","Steht der Roboter auf der 2.Pos? Mit Weiter die Sync-Position speichern","???"];
 					st_UiMsgButtons4:=["Next","Weiter","???"];
 					st_UiMsgButtons5:=["Back","Zurueck","???"];
 					st_UiMsgButtons:=["","","",st_UiMsgButtons4{n_Sp},st_UiMsgButtons5{n_Sp}];
 					st_UiMsgLines:=[st_UiMsgLine1{n_Sp},st_UiMsgLine2{n_Sp},st_UiMsgLine3{n_Sp},"",""];
					 br_UiAnswer:= UIMessageBox (\Header:=st_UiHeader{n_Sp}
									\MsgArray:=st_UiMsgLines\BtnArray:=st_UiMsgButtons\Icon:=iconInfo);
 					IF br_UiAnswer = 4 THEN
						SyncPosSetup;
					ENDIF
				ENDIF
 				GOTO ReRun2;
 			CASE 3: ! Setup, direkt anfahren
 				b_TwoSyncPos:=FALSE;
 				GOTO ReRun1;
 			CASE 4: ! Setup, auf 2 mal
 				b_TwoSyncPos:=TRUE;
 				GOTO ReRun3;
 			CASE 5: ! Setup, zurueck
 				GOTO ReRun1;
 			ENDTEST
	CASE 4: ! Anfahren
 		ReRun5:
		! Abfrage wegen Tool 0 / check because of tool zero
		IF CTool()=tool0 THEN
      		br_UiAnswer:=0;
      		st_UiHeader:=["Com, Tool check","Com, Tool Ueberpruefung","???"];
      		st_UiMsgLine1:=["Attention the active tool is tool0","Achtung das aktive Tool ist - tool0 - !!! ","???"];
      		st_UiMsgLine2:=["The robot cannot move with tool0 because","Der Roboter kann vermutlicht wegen falschen  ","???"];
      		st_UiMsgLine3:=["it has the incorrect payload configured.","Gewichtsdaten nicht bewegt werden, ","???"];
      		st_UiMsgLine4:=["Using the Jogging Window, please select the correct","bitte waehle im Bewegenfenster das richtige Tool aus,","???"];
      		st_UiMsgLine5:=["tool then press the 'Ok' button to continue.","bevor es mit Ok weiter geht.","???"];
      		st_UiMsgButtons1:=["","","???"];
      		st_UiMsgButtons2:=["","","???"];
      		st_UiMsgButtons3:=["","","???"];
      		st_UiMsgButtons4:=["Ok","Ok","???"];
      		st_UiMsgButtons5:=["","","???"];
      		st_UiMsgButtons:=[st_UiMsgButtons1{n_Sp},st_UiMsgButtons2{n_Sp},st_UiMsgButtons3{n_Sp},st_UiMsgButtons4{n_Sp},st_UiMsgButtons5{n_Sp}];
      		st_UiMsgLines:=[st_UiMsgLine1{n_Sp},st_UiMsgLine2{n_Sp},st_UiMsgLine3{n_Sp},st_UiMsgLine4{n_Sp},st_UiMsgLine5{n_Sp}];
      		!
      		br_UiAnswer:=UIMessageBox (\Header:=st_UiHeader{n_Sp}\MsgArray:=st_UiMsgLines\BtnArray:=st_UiMsgButtons\Icon:=iconWarning);
		ENDIF

        IF n_ManSyncCMD=-2 THEN
               st_UiHeader:=["Com, ManSyncIntPos","Com, ManSyncIntPos","???"];

            IF b_ManSyncInt_Found THEN
                st_UiMsgLine1:=["This Robot has the 'ManSyncIntPos' module installed","Dieser Roboeter hat das 'ManSyncIntPos' Modul installiert","???"];

                IF b_SetUpWasSelected<>TRUE THEN
                    st_UiMsgLine2:=["which may contain additional motion points which may move","welches zusaetzliche Punkte enthalten koennten, welche","???"];
                    st_UiMsgLine3:=["the robot from/to the calibration and Home1 poitions.","den Roboter von/zur Kalibrierungs und Home1 Position bewegen koennten","???"];
                    st_UiMsgLine4:=["","","???"];
                ELSE
                    st_UiMsgLine2:=["but, because the setup option was selected,","aber, da die Setup Option ausgewaehlt wurde,","???"];
                    st_UiMsgLine3:=["the positions within this module will not be executed.","werden die Positionen in diesem Modul nicht ausgefuehrt.","???"];
                    st_UiMsgLine4:=["","","???"];
                ENDIF
            ELSE
                st_UiMsgLine1:=["This Robot does not have the 'ManSyncIntPos' module installed.","Dieser Roboter hat das ManSyncIntPos Modul nicht installiert.","???"];
                st_UiMsgLine2:=["","","???"];
                st_UiMsgLine3:=["The robot will move directly to the","Der Roboter wird direkt zu den","???"];
                st_UiMsgLine4:=["predifined calibration positions.","vordefinierten Kalibrierungspositionen fahren","???"];

            ENDIF

            st_UiMsgLine5:=["Please exercise caution and watch for collisions.","Bitte vorsichtig sein und auf moegliche Kollisionen achten!","???"];

            st_UiMsgLines:=[st_UiMsgLine1{n_Sp},st_UiMsgLine2{n_Sp},st_UiMsgLine3{n_Sp},st_UiMsgLine4{n_Sp},st_UiMsgLine5{n_Sp}];

            br_UiAnswer:=UIMessageBox (\Header:=st_UiHeader{n_Sp}\MsgArray:=st_UiMsgLines\Buttons:=btnOk\Icon:=iconwarning);

            n_ManSyncCMD:=-1;

        ENDIF

 		t_Home := CTool();
 		t_home.robhold:=TRUE;
 		br_UiAnswer:=0;
 		st_UiHeader:=["Com, CalibPos","Com, Kalibrierposition","???"];
 		st_UiMsgLine1:=["The robot is at the calibration position with all axes.","Der Roboter hat die Kalibrierposition mit","???"];

        IF  b_TwoSyncPos=FALSE THEN
            IF n_ManSyncCMD=-1 AND b_ManSyncInt_Found AND b_SetUpWasSelected<>TRUE THEN
                n_ManSyncCMD:=1 ;
                %"ManSyncIntPos"%;
            ENDIF

  			MoveAbsJ jpCalibA1_A6,v200,fine,t_Home;
  			st_UiMsgLine2:=["Please check calibration marks line up.","allen Achsen erreicht, bitte alle Markierungen pruefen.","???"];
 		ELSE
 			IF 	jpCalibPos1.robax.rax_1 <> 0 OR jpCalibPos2.robax.rax_2 <> 0 OR jpCalibPos2.robax.rax_3 <> 0 OR jpCalibPos2.robax.rax_4 <> 0 OR jpCalibPos2.robax.rax_5 <> 0 OR jpCalibPos2.robax.rax_6 <> 0 THEN
				br_UiAnswer:=0;
 				st_UiHeader:=["Com, Calib Pos-Error","Com, Kalibrierposition Fehler","???"];
 				st_UiMsgLine1:=["Attention incorrect calibration position stored as at ","Achtung fehlerhafte Kalibrierposition mindestens einer Achse.","???"];
 				st_UiMsgLine2:=["least one of the axis is not at zero degrees.","Diese ist nicht auf 0 Grad in den gespeicherten Positionen.","???"];
 				st_UiMsgLine3:=["Please check positions and modify if necessary.","Beide Positionen ueberpruefen, gegebenenfalls neu speicher.","???"];
 				st_UiMsgLine4:=["The current process will be aborted.","Das Pogramm wird abgebrochen.","???"];
 				!
 				st_UiMsgButtons5:=["Abort","Abbruch","???"];
 				st_UiMsgButtons:=["","","","",st_UiMsgButtons5{n_Sp}];
 				st_UiMsgLines:=[st_UiMsgLine1{n_Sp},st_UiMsgLine2{n_Sp},st_UiMsgLine3{n_Sp},st_UiMsgLine4{n_Sp},""];
 				!
 				br_UiAnswer:=UIMessageBox (\Header:=st_UiHeader{n_Sp}\MsgArray:=st_UiMsgLines\BtnArray:=st_UiMsgButtons \Icon:=iconError);
			ENDIF

			IF br_UiAnswer=5 RETURN;

			! erste Pos von zwei
            IF n_ManSyncCMD=-1 AND b_ManSyncInt_Found AND b_SetUpWasSelected<>TRUE THEN
                n_ManSyncCMD:=2 ;
                %"ManSyncIntPos"%;
                n_ManSyncCMD:=2;
            ENDIF

			MoveAbsJ jpCalibPos1,v200,fine,t_Home;

  			st_UiMsgLine2:=["Axis 1 position reached. Please check Axis 1 calibration marks.","Achse 1 erreicht, bitte  Markierung 1 pruefen.","???"];
 			st_UiMsgButtons4:=["Next Pos 2","Weiter 2. Pos","???"];
			st_UiMsgButtons:=["","","",st_UiMsgButtons4{n_Sp},""];
			st_UiMsgLines:=[st_UiMsgLine1{n_Sp},st_UiMsgLine2{n_Sp},"","",""];
 			!
 			br_UiAnswer:=UIMessageBox (\Header:=st_UiHeader{n_Sp}\MsgArray:=st_UiMsgLines\BtnArray:=st_UiMsgButtons\Icon:=iconInfo);

            ! zweite POs

             IF n_ManSyncCMD=2 AND b_ManSyncInt_Found AND b_SetUpWasSelected<>TRUE THEN
                n_ManSyncCMD:=3 ;
                %"ManSyncIntPos"%;
            ENDIF

            MoveAbsJ jpCalibPos2,v200,fine,t_Home;

   			st_UiMsgLine2:=["Axis 2-6 & Ext axis position reached. Please check Axis 2-6 & Ext markers.","Achse 2-6 u. d. Externen erreicht, bitte Markierung 2-6 u. ext. pruefen.","???"];
		ENDIF

		st_UiMsgLine5:=["Are all the markers lined up OK?","Sind alle Markierung in Ordnung?","???"];
		!
		st_UiMsgButtons3:=["Yes","Ja","???"];
		st_UiMsgButtons4:=["No","Nein","???"];
		st_UiMsgButtons5:=["Finished","Beenden","???"];
		st_UiMsgButtons:=["","",st_UiMsgButtons3{n_Sp},st_UiMsgButtons4{n_Sp},st_UiMsgButtons5{n_Sp}];
		st_UiMsgLines:=[st_UiMsgLine1{n_Sp},st_UiMsgLine2{n_Sp},"","",st_UiMsgLine5{n_Sp}];
		!
		br_UiAnswer:=UIMessageBox (\Header:=st_UiHeader{n_Sp}\MsgArray:=st_UiMsgLines\BtnArray:=st_UiMsgButtons \Icon:=iconInfo);
		IF br_UiAnswer=5 RETURN;

        IF br_UiAnswer=4 THEN
 			br_UiAnswer:=0;
 			st_UiHeader:=["Com, CalibPos not OK","Com, Kalibrierposition n.i.O","???"];
 			st_UiMsgLine1:=["The robot is not in the correct position!","Achtung der Roboter positioniert nicht richtig!","???"];
 			st_UiMsgLine2:=["Please reset the revolution counters","Der Umdrehungszaehler der betreffenden Achsen muss ","???"];
 			st_UiMsgLine3:=["for all the axis then check the markers again.","neu gesetzt werden.","???"];
 			st_UiMsgLine4:=["","Danach die Markierung noch mal anfahren.","???"];
			!
  			st_UiMsgButtons4:=["Move again","Nochmal Anfahren","???"];
 			st_UiMsgButtons5:=["Abort","Abbruch","???"];
 			st_UiMsgButtons:=["","","",st_UiMsgButtons4{n_Sp},st_UiMsgButtons5{n_Sp}];
 			st_UiMsgLines:=[st_UiMsgLine1{n_Sp},st_UiMsgLine2{n_Sp},st_UiMsgLine3{n_Sp},st_UiMsgLine4{n_Sp},""];
 			!
 			br_UiAnswer:=UIMessageBox (\Header:=st_UiHeader{n_Sp}\MsgArray:=st_UiMsgLines\BtnArray:=st_UiMsgButtons
								\Icon:=iconError);
		ENDIF

        IF br_UiAnswer=5 RETURN;

		IF br_UiAnswer=4 THEN
			ReRun6:
			IF  b_TwoSyncPos=TRUE THEN
		  		br_UiAnswer:=0;
 				st_UiHeader:=["Com, CalibPos","Com, Kalibrierposition","???"];
 				st_UiMsgLine1:=["The Robot have two positions do you want to","Der Roboter hat 2 Positonen um die Makierungen","???"];
 				st_UiMsgLine2:=["move the robot to both or just position 2.","zu pruefen. Wollen Sie wieder beide anfahren oder nur die Zweite?","???"];
 				st_UiMsgLine3:=["","","???"];
 				st_UiMsgLine4:=["Please select.","Bitte waehlen","???"];
				!
                IF b_ManSyncInt_Found THEN
  				    st_UiMsgButtons1:=["","","???"];
                ELSE
  				    st_UiMsgButtons1:=["Both","Beide","???"];
                ENDIF
  				st_UiMsgButtons2:=["Position 2","2. Position","???"];
 				st_UiMsgButtons5:=["Abort","Abbruch","???"];
 				st_UiMsgButtons:=[st_UiMsgButtons1{n_Sp},st_UiMsgButtons2{n_Sp},"","",st_UiMsgButtons5{n_Sp}];
 				st_UiMsgLines:=[st_UiMsgLine1{n_Sp},st_UiMsgLine2{n_Sp},st_UiMsgLine3{n_Sp},st_UiMsgLine4{n_Sp},""];
 				!
 				br_UiAnswer:=UIMessageBox (\Header:=st_UiHeader{n_Sp}\MsgArray:=st_UiMsgLines\BtnArray:=st_UiMsgButtons
								\Icon:=iconInfo);
				IF br_UiAnswer=1 GOTO rerun5;
		  		IF br_UiAnswer=2 THEN

					! zweite Pos
					MoveAbsJ jpCalibPos2,v200,fine,t_Home;
					st_UiHeader:=["Com, Calibration Position","Com, Kalibrierposition","???"];
					st_UiMsgLine1:=["The robot is at the calibration position with","Der Roboter hat die Kalibrierposition mit","???"];
   					st_UiMsgLine2:=["Axis 2-6 & External position reached. Please check Axis 2-6 & Ext markers.","Achse 2-6 u. d. Externen erreicht, bitte Markierung 2-6 u. ext. pruefen.","???"];
 					st_UiMsgLine3:=["Is the Robot at the correct position?","Ist der Roboter jetzt in Ordnung?","???"];
					!
					st_UiMsgButtons3:=["Yes","Ja","???"];
					st_UiMsgButtons4:=["No","Nein","???"];
					st_UiMsgButtons5:=["Finished","Beenden","???"];
					st_UiMsgButtons:=["","",st_UiMsgButtons3{n_Sp},st_UiMsgButtons4{n_Sp},st_UiMsgButtons5{n_Sp}];
					st_UiMsgLines:=[st_UiMsgLine1{n_Sp},st_UiMsgLine2{n_Sp},st_UiMsgLine3{n_Sp},"",""];
					!
					br_UiAnswer:=UIMessageBox (\Header:=st_UiHeader{n_Sp}\MsgArray:=st_UiMsgLines\BtnArray:=st_UiMsgButtons \Icon:=iconInfo);
				ENDIF
		  		IF br_UiAnswer=4 GOTO ReRun6;
		  		IF br_UiAnswer=5 RETURN;
			ELSE
				GOTO rerun5;
			ENDIF
	    ENDIF

 		ReRun4:
 		br_UiAnswer:=0;
 		st_UiHeader:=["Com, Syncron Pos move","Com, Synch. Position fahren","???"];
 		st_UiMsgLine1:=["The robot will move to the synchronisation position","Der Roboter faehrt auf die Synchronisationsposition","???"];
 		st_UiMsgLine2:=["and will begin the soft-synchronisation function.","und startet die Soft-Synchronisierung.","???"];
 		st_UiMsgLine4:=["IMPORTANT before performing function switch to safety User.","WICHTIG Benutzerwechsel durchfuehren.","???"];
 		st_UiMsgLine5:=["This function is only permisable to safety users!","Die Synchronisierung ist nur als Safety User moeglich!","???"];
 		!
 		st_UiMsgButtons4:=["Next","Weiter","???"];
 		st_UiMsgButtons5:=["Finished","Beenden","???"];
 		st_UiMsgButtons:=["","","",st_UiMsgButtons4{n_Sp},st_UiMsgButtons5{n_Sp}];
 		st_UiMsgLines:=[st_UiMsgLine1{n_Sp},st_UiMsgLine2{n_Sp},"",st_UiMsgLine4{n_Sp},st_UiMsgLine5{n_Sp}];
 		!
 		br_UiAnswer:=UIMessageBox (\Header:=st_UiHeader{n_Sp}\MsgArray:=st_UiMsgLines\BtnArray:=st_UiMsgButtons \Icon:=iconInfo);
 		IF br_UiAnswer=5 RETURN;
 		! Synchron Pos anfahren
 		t_SMSync := CTool();
 		t_SMSync.robhold:=TRUE;

 		MoveAbsJ jpSM1SyncSwitch, v200, fine, t_SMSync;

 		! Aufruf der SM Software
 		%"SoftwareSync"%;

    	IF DOutput(SM1_do_Synced) =0 THEN
    		br_UiAnswer:=0;
    		st_UiHeader:=["Com, Error Syncron Pos","Com, Fehler Synch. Position","???"];
    		st_UiMsgLine1:=["The synchronisation has failed","Die Synchronisation ist fehlgeschlagen","???"];
    		st_UiMsgLine2:=["therefore, automatic operation is not possible.","ein Automatikbetrieb ist nicht moeglich.","???"];
    		st_UiMsgLine4:=["Eliminate the cause of the error! Then repeat the process.","Die Fehlerursache beseitigen! Danach den Vorgang wiederholen.","???"];
    		st_UiMsgButtons4:=["Retry","Wiederholen","???"];
    		st_UiMsgButtons5:=["Abort","Abbruch","???"];
    		st_UiMsgButtons:=["","","",st_UiMsgButtons4{n_Sp},st_UiMsgButtons5{n_Sp}];
    		st_UiMsgLines:=[st_UiMsgLine1{n_Sp},st_UiMsgLine2{n_Sp},"",st_UiMsgLine4{n_Sp},""];
    		!
    		br_UiAnswer:=UIMessageBox (\Header:=st_UiHeader{n_Sp}\MsgArray:=st_UiMsgLines\BtnArray:=st_UiMsgButtons \Icon:=iconError);
    		IF br_UiAnswer=4 GOTO ReRun4;
        ELSE
 			br_UiAnswer:=0;
 			st_UiHeader:=["Com, Robot Synchron","Com, Roboter Synchron ","???"];
 			st_UiMsgLine1:=["The Robot is synchronised.","Der Roboter ist synchronisiert.","???"];
  			st_UiMsgButtons4:=["Check Brake","Bremsen testen","???"];
 			st_UiMsgButtons5:=["Finished","Beenden","???"];
			st_UiMsgButtons:=["","","",st_UiMsgButtons4{n_Sp},st_UiMsgButtons5{n_Sp}];
			st_UiMsgLines:=[st_UiMsgLine1{n_Sp},"","","",""];
 			!
 			br_UiAnswer:=UIMessageBox (\Header:=st_UiHeader{n_Sp}\MsgArray:=st_UiMsgLines\BtnArray:=st_UiMsgButtons \Icon:=iconInfo);
			!
			IF br_UiAnswer=4  THEN
				jpTempPos := CJointT();
                br_UiAnswer:=0;

				WHILE ABS(jpTempPos.extax.eax_a) <= 5 AND br_UiAnswer<>4 DO
				 	br_UiAnswer:=0;
 					st_UiHeader:=["Com, Brake Test","Com, Bremsentest","???"];
 					st_UiMsgLine1:=["Warning! The Linear track axis 7 is near 0mm and may fail braketest.","Achtung, die Achse 7 ist nahe 0 mm der Bremsentest koennte fehlschlagen","???"];

 					st_UiMsgLine3:=["Select 'Ignore' to start the Brake Test at current position.","Mit 'ignorieren' wird der Bremsentest in der aktuellen Position gestartet.","???"];
 					st_UiMsgLine4:=["Select 'Jog' then please move the axis >5 mm then 'Play' to start test.","Mit 'Jog' Bitte die Achse min. >5 mm. bewegen, mit 'Play' Test starten","???"];

                    st_UiMsgButtons4:=["Ignore","ignorieren","???"];
  					st_UiMsgButtons5:=["Jog","Jog","???"];

					st_UiMsgButtons:=["","","",st_UiMsgButtons4{n_Sp},st_UiMsgButtons5{n_Sp}];
					st_UiMsgLines:=[st_UiMsgLine1{n_Sp},"",st_UiMsgLine3{n_Sp},st_UiMsgLine4{n_Sp},""];

 					br_UiAnswer:=UIMessageBox (\Header:=st_UiHeader{n_Sp}\MsgArray:=st_UiMsgLines\BtnArray:=st_UiMsgButtons \Icon:=iconError);

                    IF br_UiAnswer=5 THEN
                        ClearPath;
                        Stop;
                    ENDIF

                    jpTempPos := CJointT();
                ENDWHILE

                CyclicBrakeCheck_V2;

			ENDIF
 		ENDIF

        IF n_ManSyncCMD=0 AND b_ManSyncInt_Found AND b_SetUpWasSelected<>TRUE THEN

            st_UiHeader:=["Com, ManSyncIntPos","Com, ManSyncIntPos","???"];
            st_UiMsgLine1:=["This Robot will move back to the Home Position 1.","Dieser Roboter wird zurueck zur Home Position 1 fahren.","???"];
            st_UiMsgLine2:=["","","???"];
            st_UiMsgLine3:=["","","???"];
            st_UiMsgLine4:=["","","???"];
            st_UiMsgLine5:=["","","???"];

            st_UiMsgLines:=[st_UiMsgLine1{n_Sp},st_UiMsgLine2{n_Sp},st_UiMsgLine3{n_Sp},st_UiMsgLine4{n_Sp},st_UiMsgLine5{n_Sp}];

            br_UiAnswer:=UIMessageBox (\Header:=st_UiHeader{n_Sp}\MsgArray:=st_UiMsgLines\Buttons:=btnOk\Icon:=iconwarning);

     		n_ManSyncCMD:=4 ;
            %"ManSyncIntPos"%;
        ENDIF
 CASE 5: ! Abbruch
 	TPErase;
 	RETURN;
 ENDTEST
 !
 TPErase;

 ERROR
!** Error Handler**

SkipWarn;
TEST ERRNO

CASE ERR_REFUNKPRC:
    IF n_ManSyncCMD=-2 THEN
        b_ManSyncInt_Found:=FALSE ;
        TRYNEXT;
    ENDIF

ENDTEST

ENDPROC ! ManSyncService ()

!*******************************************************************************

PROC PLC_Release (string Comment \VAR signaldo Set_ \VAR signaldi Wait_ \switch InPos\num Job)
 !****************************************
 !* Request operation handshake with PLC *
 !****************************************

 VAR errnum errno1;
 VAR signaldo PLC_JobStarted;
 VAR string st_alias;
 CONST string st_C:="PLC_do_Job";
 CONST string st_D:="_Started";

 IF Present(Job) CheckValue Job, 1, 32, 0, "Job Number";

 ! Abfrage fuer das Argument InPos
 IF Present (Inpos) WaitRob \InPos;

 ! Setzendes des Ausgangs

 IF Present (Set_) Set Set_;
 ! Warten auf die rueckmeldung von der SPS

 IF Present(Wait_) WaitDI Wait_,1\MaxTime:=3;
 !****************************
 !* Waiting PLC reease Input *
 !****************************

 IF Present(Job) THEN
	! Signalnamen erzeugen / signalname to procreate
	IF Job <10 THEN
		st_alias :=st_C+"0"+NumToStr(Job,0)+st_D;
	ELSE
		st_alias :=st_C+NumToStr(Job,0)+st_D;
	ENDIF

	AliasIO st_alias, PLC_JobStarted;

  	Set PLC_JobStarted;
 ENDIF

  ! Ruecksetzen des Ausgangs
 IF  Present (Set_) AND Present(Wait_) Reset Set_;

 ERROR
 !** Error Handler**
 SkipWarn;

 MsgBox_Clear;

 TEST ERRNO
 CASE ERR_WAIT_MAXTIME:
	st_UiHeader:=["PLC_Release, Waiting!!","PLC_Release, Warte auf ...","???"];
	st_UiMsgLine2:=["Waiting for "+ArgName(Wait_)+":= 1","Warte auf "+ArgName(Wait_)+":= 1","???"];

    IF Present(Set_) THEN
        st_UiMsgLine4:=["The Output '"+ArgName(Set_)+"' was set but, the robot","Der Ausgang "+ArgName(Set_)+" wurde gesetzt.","???"];
        st_UiMsgLine5:=["is waiting for the release signal '"+ArgName(Wait_)+"' from the PLC.","Der Roboter wartet auf die Freigabe von "+ArgName(Wait_)+" durch die SPS.","???"];
    ELSE
         st_UiMsgLine5:=["Robot is waiting for the release signal '"+ArgName(Wait_)+"' from the PLC.","Der Roboter wartet auf die Freigabe von "+ArgName(Wait_)+" durch die SPS.","???"];
    ENDIF

    UIMsgBox\Header:=st_UiHeader{n_Sp},Comment \MsgLine2:=st_UiMsgLine2{n_Sp}\MsgLine4:=st_UiMsgLine4{n_Sp}
					\MsgLine5:=st_UiMsgLine5{n_Sp}\Buttons:=btnNone\Icon:=iconInfo\DIBreak:=Wait_
					\BreakFlag:=errno1;
	TRYNEXT;

 ENDTEST
ENDPROC ! PLC_Release()

!*******************************************************************************

PROC MsgBox(\VAR signaldi diBreakSignal\VAR signaldo doBreakSignal\string Line1\string Line2\switch ErrorToPLC |switch StopToPLC)
 !*****************************************************************************************************
 !*                             Prozedur meldet Meldung/Fehler an die SPS und                         *
 !*                      Zeigt Fehler auf dem TP und wartet auf eine Aktion vom Bediener              *
 !*                                                                                                   *
 !* optionale Parameter: \VAR signaldi diBreakSignal = Abbruchsignal zum abloeschen der Meldung am TP  *
 !*						\VAR signaldi doBreakSignal = Abbruchsignal zum abloeschen der Meldung am TP  *
 !*						\string Line1 = Es wird der uebergebene Text in Line1 angezeigt               *
 !*						\string Line2 = Es wird der uebergebene Text in Line2 angezeigt               *
 !*						\switch ErrorToPLC) = Es wird der Ausgang PLC_do_ErrorToPLC 1                *
 !*						|switch StopToPLC) = Es wird der Ausgang PLC_do_StopToPLC 1                  *
 !*                                                                                                   *
 !*                          Message handler logs / errors to the PLC, and                            *
 !*                  Displays error on TP and waits for an action by the operator                     *
 !*****************************************************************************************************
 VAR errnum errno1;
 CONST string st_MsgBoxLine1{3}:=["Waiting for: ","Warte auf: ","???"];
 CONST string st_MsgBoxLine2{3}:=["Error: ","Fehler: ","???"];
 VAR string st_MsgBoxLine_1;
 VAR string st_MsgBoxLine_2;
 VAR string st_MsgBox_buttons{5};
 VAR string st_MsgBoxLine1_5{5};
 VAR bool b_Timeflag:=FALSE;
 VAR icondata id_MsgIcon;
 VAR signaldo alias_do;
 VAR signaldi alias_di;
 VAR bool b_IO_RequiredStateOK:=TRUE;
 VAR bool b_IO_Defined:=TRUE;
 VAR dionum dn_State_Required;

 n_MsgBoxAnswer:=0;
 IF Present(Line1) THEN
 	st_MsgBoxLine_1:=Line1;
 ELSE
 	IF st_MsgBoxSignalValue <> stEmpty THEN
 		st_MsgBoxLine_1:=st_MsgBoxLine1{n_Sp}+st_MsgBoxSignal+"= "+st_MsgBoxSignalValue;
 	ELSE
 		st_MsgBoxLine_1:=st_MsgBoxLine1{n_Sp}+st_MsgBoxSignal;
 	ENDIF
 ENDIF

 IF Present(Line2) THEN
 	st_MsgBoxLine_2:=Line2;
 ELSE
 	IF n_MsgBoxApplError > 0 THEN
 		st_MsgBoxLine_2:=st_MsgBoxLine2{n_Sp}+st_MsgBoxGeraeteName{n_Sp}+" "+NumToStr(n_MsgBoxGeraeteNr,0)
 		+" Error Code: "+NumToStr(n_MsgBoxApplError,0);
 	ELSE
 		st_MsgBoxLine_2:=st_MsgBoxLine2{n_Sp}+st_MsgBoxGeraeteName{n_Sp}+" "+NumToStr(n_MsgBoxGeraeteNr,0);
 	ENDIF
 ENDIF
 ErrWrite \W,	st_MsgBoxHeader{n_Sp},st_MsgBoxLine_1\
 RL2:=st_MsgBoxLine_2\
 RL3:=" "\
 RL4:=st_MsgBoxElogLine4+"/"+NumToStr(n_Step,0)+"/"+NumToStr(n_MsgBoxApplError,0)+"/"+NumToStr(n_MsgBoxPLC_Error,0);
 !
 ! Icon vorbesetzen / Text from Icon
 id_MsgIcon:=iconInfo;
 IF Present(ErrorToPLC) id_MsgIcon:=iconWarning;
 IF Present(StopToPLC)  id_MsgIcon:=iconError;
 ! Wenn ErrorNr >0 oder kein Hinergrundtask dann setze Fehler zur SPS ab /
 ! If ErrorNr> 0, or no errors in ground task then dont send errors to the PLC
 IF n_MsgBoxPLC_Error  >0 AND TaskRunRob( )THEN
	!Fehlernummer zur SPS setzen / Error number send to the PLC
	SetGO PLC_go_ErrCode, n_MsgBoxPLC_Error;
	! setze Fehlerart\Send fault control bit
	IF Present(ErrorToPLC) THEN
		Set PLC_do_ErrorToPLC;
	ELSEIF Present (StopToPLC)THEN
		Set PLC_do_StopToPLC;
	ELSE
		Set PLC_do_MsgToPLC;
	ENDIF
	!
 ENDIF
 !
 st_MsgBoxLine1_5:=[st_MsgBoxLine_1,st_MsgBoxLine_2,st_MsgBoxLine3{n_Sp},st_MsgBoxLine4{n_Sp},st_MsgBoxLine5{n_Sp}];
 st_MsgBox_buttons:=[st_MsgBoxbutton1{n_Sp},st_MsgBoxbutton2{n_Sp},st_MsgBoxbutton3{n_Sp},st_MsgBoxbutton4{n_Sp},st_MsgBoxbutton5{n_Sp}];
 !
 IF Present(diBreakSignal) AND Present(doBreakSignal) THEN
 	WaitUntil diBreakSignal=0 AND DOutput(doBreakSignal) = 0\MaxTime:=2\TimeFlag:=b_Timeflag;
 	n_MsgBoxAnswer:= UIMessageBox (\Header:=st_MsgBoxHeader{n_Sp}\MsgArray:=st_MsgBoxLine1_5\
 												BtnArray:=st_MsgBox_buttons\Icon:=id_MsgIcon\DIBreak:=diBreakSignal\
 												DOBreak:=doBreakSignal\BreakFlag:=errno1);
 ELSEIF Present(diBreakSignal) THEN
 	WaitDI diBreakSignal,0\MaxTime:=2\TimeFlag:=b_Timeflag;
 	n_MsgBoxAnswer:= UIMessageBox (\Header:=st_MsgBoxHeader{n_Sp}\MsgArray:=st_MsgBoxLine1_5\
 												BtnArray:=st_MsgBox_buttons\Icon:=id_MsgIcon\
 												DIBreak:=diBreakSignal\BreakFlag:=errno1);
 ELSEIF Present(doBreakSignal) THEN
 	WaitDO doBreakSignal,0\MaxTime:=2\TimeFlag:=b_Timeflag;
 	n_MsgBoxAnswer:= UIMessageBox (\Header:=st_MsgBoxHeader{n_Sp}\MsgArray:=st_MsgBoxLine1_5\
 												BtnArray:=st_MsgBox_buttons\Icon:=id_MsgIcon\
 												DOBreak:=doBreakSignal\BreakFlag:=errno1);
 ELSE
 	n_MsgBoxAnswer:= UIMessageBox (\Header:=st_MsgBoxHeader{n_Sp}\MsgArray:=st_MsgBoxLine1_5\
 												BtnArray:=st_MsgBox_buttons\Icon:=id_MsgIcon\BreakFlag:=errno1);
 ENDIF

 !Code to avoid error code being reset when signal message box is waiting is still in incorrect state
 IF Present(ErrorToPLC) AND StrLen(st_MsgBoxSignal)>4 AND StrLen(st_MsgBoxSignalValue)=1 THEN

    IF StrMatch (st_MsgBoxSignal,1," ") = StrLen(st_MsgBoxSignal)+1 AND (st_MsgBoxSignalValue="0" OR st_MsgBoxSignalValue="1") THEN

        IF st_MsgBoxSignalValue="0" THEN
            dn_State_Required:=0;
        ELSE
            dn_State_Required:=1;
        ENDIF

        IF StrMatch(st_MsgBoxSignal,1,"_di_") <> StrLen(st_MsgBoxSignal)+1 THEN
            AliasIO st_MsgBoxSignal, alias_di;

            IF b_IO_Defined THEN
                b_IO_RequiredStateOK:= (alias_di=dn_State_Required);
            ENDIF

        ELSEIF StrMatch(st_MsgBoxSignal,1,"_do_") <> StrLen(st_MsgBoxSignal)+1 THEN
            AliasIO st_MsgBoxSignal, alias_do;

            IF b_IO_Defined THEN
                b_IO_RequiredStateOK:= (DOutput(alias_do)= dn_State_Required);
            ENDIF
         ENDIF
    ENDIF
ENDIF


 IF n_MsgBoxPLC_Error >0 THEN
     IF b_IO_RequiredStateOK THEN
         SetGO PLC_go_ErrCode, 0;
         Reset PLC_do_ErrorToPLC;
         n_PLC_ErrCode_Mem:=-2;
     ELSE
        n_PLC_ErrCode_Mem:=n_MsgBoxPLC_Error;
     ENDIF

 	Reset PLC_do_MsgToPLC;
 	Reset PLC_do_StopToPLC;
 ENDIF
 !
 MsgBox_Clear;
 TPShow TP_LATEST;

 ERROR
!** Error Handler **

TEST ERRNO

CASE ERR_ALIASIO_DEF,ERR_ALIASIO_TYPE:
    b_IO_Defined:=FALSE;
    TRYNEXT;
ENDTEST

ENDPROC !(MsgBox)

!*******************************************************************************

PROC MsgBox_Clear ()
!**********************************
!*    Messagebox clear routine    *
!**********************************

 !Reset st VAR
 st_MsgBoxHeader:=["","",""];
 st_MsgBoxLine3:=["","",""];
 st_MsgBoxLine4:=["","",""];
 st_MsgBoxLine5:=["","",""];
 !Reset Tasten 1-5
 st_MsgBoxbutton1:=["","",""];
 st_MsgBoxbutton2:=["","",""];
 st_MsgBoxbutton3:=["","",""];
 st_MsgBoxbutton4:=["","",""];
 st_MsgBoxbutton5:=["","",""];
 !Reset st
 st_MsgBoxGeraeteName:=["","",""];
 n_MsgBoxGeraeteNr:=0;
 st_MsgBoxSignal:="";
 n_MsgBoxApplError:=0;
 n_MsgBoxPLC_Error:=0;
 st_MsgBoxElogLine4:="";
ENDPROC !(MsgBox_Clear)

!*******************************************************************************

PROC MsgBoxEv(\VAR signaldi diBreakSignal\VAR signaldo doBreakSignal\string Line1\string Line2\switch ErrorToPLC |switch StopToPLC)
 !*****************************************************************************************************
 !*                             Prozedur meldet Meldung/Fehler von einer Eventrout. an die SPS und    *
 !*                      Zeigt Fehler auf dem TP und wartet auf eine Aktion vom Bediener              *
 !*                                                                                                   *
 !* optionale Parameter: \VAR signaldi diBreakSignal = Abbruchsignal zum abloeschen der Meldung am TP  *
 !*						\VAR signaldi doBreakSignal = Abbruchsignal zum abloeschen der Meldung am TP  *
 !*						\string Line1 = Es wird der uebergebene Text in Line1 angezeigt               *
 !*						\string Line2 = Es wird der uebergebene Text in Line2 angezeigt               *
 !*						\switch ErrorToPLC) = Es wird der Ausgang PLC_do_ErrorToPLC 1                *
 !*						|switch StopToPLC) = Es wird der Ausgang PLC_do_StopToPLC 1                  *
 !*                                                                                                   *
 !*                          Message handler logs / errors from Eventrout. to the PLC, and                            *
 !*                  Displays error on TP and waits for an action by the operator                     *
 !*****************************************************************************************************
 VAR errnum errno1;
 CONST string st_MsgBoxEvLine1{3}:=["Waiting for: ","Warte auf: ","???"];
 CONST string st_MsgBoxEvLine2{3}:=["Error: ","Fehler: ","???"];
 VAR string st_MsgBoxEvLine_1;
 VAR string st_MsgBoxEvLine_2;
 VAR string st_MsgBoxEv_buttons{5};
 VAR string st_MsgBoxEvLine1_5{5};
 VAR bool b_Timeflag:=FALSE;
 VAR icondata id_MsgBoxEvIcon;
 VAR dionum dn_PLC_do_MsgToPLC:=0;
 VAR dionum dn_PLC_do_ErrorToPLC:=0;
 VAR dionum dn_PLC_do_StopToPLC:=0;
 !
 n_MsgBoxEvAnswer:=0;
 IF Present(Line1) THEN
 	st_MsgBoxEvLine_1:=Line1;
 ELSE
 	IF st_MsgBoxEvSignalValue <> stEmpty THEN
 		st_MsgBoxEvLine_1:=st_MsgBoxEvLine1{n_Sp}+st_MsgBoxEvSignal+"= "+st_MsgBoxEvSignalValue;
 	ELSE
 		st_MsgBoxEvLine_1:=st_MsgBoxEvLine1{n_Sp}+st_MsgBoxEvSignal;
 	ENDIF
 ENDIF
 IF Present(Line2) THEN
 	st_MsgBoxEvLine_2:=Line2;
 ELSE
 	IF n_MsgBoxEvApplError > 0 THEN
 		st_MsgBoxEvLine_2:=st_MsgBoxEvLine2{n_Sp}+st_MsgBoxEvGeraeteName{n_Sp}+" "+NumToStr(n_MsgBoxEvGeraeteNr,0)
 		+" Error Code: "+NumToStr(n_MsgBoxEvApplError,0);
 	ELSE
 		st_MsgBoxEvLine_2:=st_MsgBoxEvLine2{n_Sp}+st_MsgBoxEvGeraeteName{n_Sp}+" "+NumToStr(n_MsgBoxEvGeraeteNr,0);
 	ENDIF
 ENDIF
  ErrWrite \W,	st_MsgBoxEvHeader{n_Sp},st_MsgBoxEvLine_1\
  RL2:=st_MsgBoxEvLine_2\
  RL3:=" "\
  RL4:=st_MsgBoxEvElogLine4+"/"+NumToStr(n_Step,0)+"/"+NumToStr(n_MsgBoxEvApplError,0)+"/"
  +NumToStr(n_MsgBoxEvPLC_Error,0);
 !
 ! Icon vorbesetzen
  id_MsgBoxEvIcon:=iconInfo;
  IF Present(ErrorToPLC) id_MsgBoxEvIcon:=iconWarning;
  IF Present(StopToPLC)  id_MsgBoxEvIcon:=iconError;
  ! Wenn ErrorNr >0 oder kein Hintergrundtask dann setze Fehler zur SPS ab
 IF n_MsgBoxEvPLC_Error  >0 AND TaskRunRob( )THEN
  !
  IF DOutput(PLC_do_MsgToPLC) = 1 dn_PLC_do_MsgToPLC:=1;
  IF DOutput(PLC_do_ErrorToPLC) = 1 dn_PLC_do_ErrorToPLC:=1;
  IF DOutput(PLC_do_StopToPLC) = 1 dn_PLC_do_StopToPLC:=1;
  SetGO PLC_go_ErrCode, 0;
  Reset PLC_do_MsgToPLC;
  Reset PLC_do_ErrorToPLC;
  Reset PLC_do_StopToPLC;
  !
   !Fehlernummer zur SPS setzen
   SetGO PLC_go_ErrCode, n_MsgBoxEvPLC_Error;
   ! setze Fehlerart
  IF Present(ErrorToPLC) THEN
   Set PLC_do_ErrorToPLC;
  ELSEIF Present (StopToPLC)THEN
   Set PLC_do_StopToPLC;
  ELSE
   Set PLC_do_MsgToPLC;
  ENDIF
 !
 ENDIF
 !
 st_MsgBoxEvLine1_5:=[st_MsgBoxEvLine_1,st_MsgBoxEvLine_2,st_MsgBoxEvLine3{n_Sp},st_MsgBoxEvLine4{n_Sp},st_MsgBoxEvLine5{n_Sp}];
 st_MsgBoxEv_buttons:=[st_MsgBoxEvbutton1{n_Sp},st_MsgBoxEvbutton2{n_Sp},st_MsgBoxEvbutton3{n_Sp},st_MsgBoxEvbutton4{n_Sp},st_MsgBoxEvbutton5{n_Sp}];
 !
 IF Present(diBreakSignal) AND Present(doBreakSignal) THEN
 		WaitUntil diBreakSignal=0 AND DOutput(doBreakSignal) = 0\MaxTime:=2\TimeFlag:=b_Timeflag;
 		n_MsgBoxEvAnswer:= UIMessageBox (\Header:=st_MsgBoxEvHeader{n_Sp}\MsgArray:=st_MsgBoxEvLine1_5\
 													BtnArray:=st_MsgBoxEv_buttons\Icon:=id_MsgBoxEvIcon\
 													DIBreak:=diBreakSignal\	DOBreak:=doBreakSignal\
 	           										BreakFlag:=errno1);
 ELSEIF Present(diBreakSignal) THEN
 		WaitDI diBreakSignal,0\MaxTime:=2\TimeFlag:=b_Timeflag;
 		n_MsgBoxEvAnswer:= UIMessageBox (\Header:=st_MsgBoxEvHeader{n_Sp}\MsgArray:=st_MsgBoxEvLine1_5\
 													BtnArray:=st_MsgBoxEv_buttons\Icon:=id_MsgBoxEvIcon\
 													DIBreak:=diBreakSignal\BreakFlag:=errno1);
 ELSEIF Present(doBreakSignal) THEN
 		WaitDO doBreakSignal,0\MaxTime:=2\TimeFlag:=b_Timeflag;
 		n_MsgBoxEvAnswer:= UIMessageBox (\Header:=st_MsgBoxEvHeader{n_Sp}\MsgArray:=st_MsgBoxEvLine1_5\
 													BtnArray:=st_MsgBoxEv_buttons\Icon:=id_MsgBoxEvIcon\
 													DOBreak:=doBreakSignal\BreakFlag:=errno1);
 ELSE
 		n_MsgBoxEvAnswer:= UIMessageBox (\Header:=st_MsgBoxEvHeader{n_Sp}\MsgArray:=st_MsgBoxEvLine1_5\
 													BtnArray:=st_MsgBoxEv_buttons\Icon:=id_MsgBoxEvIcon\
 	           										BreakFlag:=errno1);
 ENDIF
 !
 IF n_MsgBoxEvPLC_Error >0 THEN
 	SetGO PLC_go_ErrCode, n_MsgBoxPLC_Error;
 	SetDO PLC_do_MsgToPLC, dn_PLC_do_MsgToPLC;
 	SetDO PLC_do_ErrorToPLC, dn_PLC_do_ErrorToPLC;
 	SetDO PLC_do_StopToPLC, dn_PLC_do_StopToPLC;
 ENDIF
 MsgBoxEv_Clear;
 TPShow TP_LATEST;
 !
ENDPROC !(MsgBoxEv)

!*******************************************************************************

PROC MsgBoxEv_Clear()
!**********************************
!* Messagebox event clear routine *
!**********************************

 !Reset st VAR	MsgBoxEv
 st_MsgBoxEvHeader:=["","",""];
 st_MsgBoxEvLine3:=["","",""];
 st_MsgBoxEvLine4:=["","",""];
 st_MsgBoxEvLine5:=["","",""];
 !Reset Tasten 1-5
 st_MsgBoxEvbutton1:=["","",""];
 st_MsgBoxEvbutton2:=["","",""];
 st_MsgBoxEvbutton3:=["","",""];
 st_MsgBoxEvbutton4:=["","",""];
 st_MsgBoxEvbutton5:=["","",""];
 !Reset st
 st_MsgBoxEvGeraeteName:=["","",""];
 n_MsgBoxEvGeraeteNr:=0;
 st_MsgBoxEvSignal:="";
 n_MsgBoxEvApplError:=0;
 n_MsgBoxEvPLC_Error:=0;
 st_MsgBoxEvElogLine4:="";
ENDPROC ! (MsgBoxEv_Clear)

!*******************************************************************************


PROC MsgBoxBreak (string SignalName,dNum RequiredValue,\SWITCH InverseControl)
!*******************************************************************
!*  Procedure for the Msgbox function to allow the Break function  *
!*      to operate for a signal that goes from High to Low.        *
!*           Software works in association with TB_COM             *
!*******************************************************************

VAR Bool b_Timeout;
VAR String st_Temp;

!Transfer to Persistent string
st_MsgboxBrk_SignalName:=SignalName;
dn_MsgboxBrk_ReqValue:=RequiredValue;
b_Invert_Control:=Present(InverseControl);

!Reset TB_Com Return String
st_MsgboxBrk_ReturnName:=" ";

WHILE st_MsgboxBrk_SignalName<>st_MsgboxBrk_ReturnName DO

      WaitUntil st_MsgboxBrk_SignalName=st_MsgboxBrk_ReturnName\MaxTime:=5 \TimeFlag:=b_Timeout;
      !**************************************
      !* Waiting for the TB_Com routine to  *
      !*  echo back the string sent to it.  *
      !**************************************

      IF b_Timeout THEN
            TPErase;
            st_MsgBoxHeader:=["MsgBoxIBreak Error" ,"MsgBoxIBreak Error","???"];

            IF st_MsgboxBrk_SignalName="SignalNameError" THEN
                  st_MsgBoxLine3:=["The Signal name programmed '" + SignalName + "' is invalid." ,"Der Signal namen programmiert '" + SignalName + "' ist ungültig.","???"];
                  st_MsgBoxLine5:=["Please Select 'OK' to Retry.","Bitte wählen Sie 'OK' zu wiederholen.","???"];
                  n_MsgBoxAnswer:= UIMessageBox (\Header:=st_MsgBoxHeader{n_Sp}\MsgArray:=[" "," ",st_MsgBoxLine3{n_Sp},st_MsgBoxLine4{n_Sp},st_MsgBoxLine5{n_Sp}]\Buttons:=btnOK\Icon:=iconError);
                  Stop;
            ELSE
                  st_MsgBoxLine3:=["TB Com Communication Timeout." ,"TB Com Communication Timeout.","???"];
                  st_MsgBoxLine5:=["Please Select 'OK' to Retry.","Bitte wählen Sie 'OK' zu wiederholen.","???"];
                  n_MsgBoxAnswer:= UIMessageBox (\Header:=st_MsgBoxHeader{n_Sp}\MsgArray:=[" "," ",st_MsgBoxLine3{n_Sp},st_MsgBoxLine4{n_Sp},st_MsgBoxLine5{n_Sp}]\Buttons:=btnOK\Icon:=iconError);
            ENDIF

      ENDIF
ENDWHILE

ENDPROC !(MsgBoxBreak)


!*******************************************************************************


PROC Log_Message (string Category, string Message,\Num TimeOut)
!************************************************
!*   Send message TXT data to log file system   *
!************************************************
VAR bool b_timeout;
VAR num nTimeout:=0;

IF Present(TimeOut) THEN
    IF TimeOut<0 OR TimeOut>5 TimeOut:=0;
    nTimeout:=TimeOut;
ENDIF

WaitUntil s_LOG_TX_Data=""\Maxtime:=nTimeOut\TimeFlag := b_timeout;
!*****************************************************
!* Waiting for message to be written to log database *
!*****************************************************

s_LOG_TX_Cat:=Category;
s_LOG_TX_Data:=Message;

ENDPROC !(Log_Message)


!*******************************************************************************


FUNC Num GetGroupIP (VAR Signaldi diSignalName,Num n_diBitLength)
!***************************************
!* Procedure to return a numeric value *
!*    from a group of Digital Inputs   *
!***************************************

VAR signaldi di_Temp;

VAR Num n_FirstBitNr;
VAR Num n_LastBitNr;
VAR Num n_diSignal_Length;
VAR Num n_CharNr;
VAR Num n_ScrollNr;
VAR Num n_ValueCount;
VAR Num n_CharFirstNumber;
VAR Num n_CharLastNumber;
VAR Num n_CharNumberCount;
VAR Num n_NumberCharlength;

VAR String st_diSignalName;
VAR String st_FirstbitNr;
VAR String st_diSignalDesc;
VAR String st_diSignalDesc1;
VAR String st_diSignalDesc2;
VAR String st_tempString ;

!Stop advance pointer
WaitTime\Inpos, 0.0 ;

!Check first bit configured is a valid input
st_diSignalName:=ArgName(diSignalName);
AliasIO st_diSignalName, di_Temp;

!Check input name length
n_diSignal_Length:=StrLen(st_diSignalName);

IF n_diSignal_Length > 3 THEN
	!Determine which characters the Bit numbers start
	n_CharFirstNumber:=StrFind(st_diSignalName,1,STR_DIGIT) ;

	!Determine how many characters are numeric
	IF n_CharFirstNumber<n_diSignal_Length THEN
		n_CharLastNumber:=StrFind(st_diSignalName,n_CharFirstNumber+1,STR_DIGIT);
	ELSE
		n_CharLastNumber:=n_diSignal_Length;
	ENDIF

	n_NumberCharlength:=n_CharLastNumber-n_CharFirstNumber +1;

	!Check that there are numbers in signal description
	WHILE n_CharFirstNumber>n_diSignal_Length DO
		TPErase;
		st_MsgBoxHeader:=["GetGIValue  Signal=" + st_diSignalName ,"GetGIValue  Signal=" + st_diSignalName,"???"];
		st_MsgBoxLine3:=["There are no bit numbers in the signal name defined." ,"Es gibt keine Bit-Zahlen in der Signal-Namen definiert","???"];
		st_MsgBoxLine4:=["Please check Configuration.","Bitte Überprüfe Konfiguration.","???"];
		n_MsgBoxAnswer:= UIMessageBox (\Header:=st_MsgBoxHeader{n_Sp}\MsgArray:=[" "," ",st_MsgBoxLine3{n_Sp},st_MsgBoxLine4{n_Sp}," "]\Buttons:=btnOK\Icon:=iconError) ;

		STOP;
	ENDWHILE

	n_CharNumberCount:=1;

	!Check how many characters are numbers
	FOR n_CharNr FROM n_CharFirstNumber +1 TO n_diSignal_Length DO
		IF StrFind(st_diSignalName,n_CharNr,STR_DIGIT)<=n_diSignal_Length THEN
			INCR n_CharNumberCount ;
		ENDIF
	ENDFOR

	!Check that there are no more than 3 numbers in the signal description
	WHILE n_CharNumberCount>2 DO
		TPErase;
		st_MsgBoxHeader:=["GetGIValue  Signal=" + st_diSignalName ,"GetGIValue  Signal=" + st_diSignalName,"???"];
		st_MsgBoxLine3:=["There are more than two numbers in the" ,"Es gibt mehr als zwei Zahlen in der","???"];
		st_MsgBoxLine4:=["signal name defined. Check Configuration.","Signal-Name definiert. Konfiguration prüfen.","???"];
		n_MsgBoxAnswer:= UIMessageBox (\Header:=st_MsgBoxHeader{n_Sp}\MsgArray:=[" "," ",st_MsgBoxLine3{n_Sp},st_MsgBoxLine4{n_Sp}," "]\Buttons:=btnOK\Icon:=iconError) ;

		STOP;
	ENDWHILE

	!Check that there are no less than numbers in signal description
	WHILE n_CharNumberCount<2 DO
		TPErase;
		st_MsgBoxHeader:=["GetGIValue  Signal=" + st_diSignalName ,"GetGIValue  Signal=" + st_diSignalName,"???"];
		st_MsgBoxLine3:=["The are less than two numbers in the" ,"Das sind weniger als zwei Zahlen in der","???"];
		st_MsgBoxLine4:=["signal name defined. Check Configuration.","Signal-Name definiert. Konfiguration prüfen.","???"];
		n_MsgBoxAnswer:= UIMessageBox (\Header:=st_MsgBoxHeader{n_Sp}\MsgArray:=[" "," ",st_MsgBoxLine3{n_Sp},st_MsgBoxLine4{n_Sp}," "]\Buttons:=btnOK\Icon:=iconError) ;

		STOP;
	ENDWHILE

	!Get Bit number as a string
	st_FirstbitNr:=StrPart(st_diSignalName,n_CharFirstNumber,n_NumberCharlength);

	!Check st_FirstbitNr is a number
	WHILE StrToVal(st_FirstbitNr,n_FirstBitNr)<>TRUE DO
		TPErase;
		st_MsgBoxHeader:=["GetGIValue  Signal=" + st_diSignalName ,"GetGIValue  Signal=" + st_diSignalName ,"???"];
		st_MsgBoxLine3:=["There are not two consecutive bit numbers defined." ,"Es gibt nicht zwei aufeinander folgenden Bit-Zahlen definiert.","???"];
		st_MsgBoxLine4:=["Please Check Configuration.","Bitte Überprüfe Konfiguration.","???"];
		n_MsgBoxAnswer:= UIMessageBox (\Header:=st_MsgBoxHeader{n_Sp}\MsgArray:=[" "," ",st_MsgBoxLine3{n_Sp},st_MsgBoxLine4{n_Sp}," "]\Buttons:=btnOK\Icon:=iconError) ;

		STOP;
	ENDWHILE

	st_diSignalDesc1:=StrPart(st_diSignalName,1,n_CharFirstNumber-1);

	IF (n_CharFirstNumber+1)=n_diSignal_Length OR n_CharFirstNumber=n_diSignal_Length THEN
		!Bit numbers are the last or last two characters
		st_diSignalDesc2:="" ;
		st_diSignalDesc:=st_diSignalDesc1 + "??" ;
	ELSE
		st_diSignalDesc2:=StrPart(st_diSignalName,n_CharFirstNumber+2,n_diSignal_Length-n_CharFirstNumber-1);
		st_diSignalDesc:=st_diSignalDesc1 + "??" + st_diSignalDesc2 ;
	ENDIF

	n_LastBitNr:=n_FirstBitNr+n_diBitLength-1;

	IF n_diBitLength<1 OR n_diBitLength>16 THEN
		!Check n_diBitLength paramater is valid

		WHILE TRUE DO
			TPErase;
			st_MsgBoxHeader:=["GetGIValue Signal=" + st_diSignalDesc ,"GetGIValue Signal=" + st_diSignalDesc,"???"];
			st_MsgBoxLine3:=["The Bit length Specified=" + ValToStr(n_diBitLength) + ". Value must be between 1-16." ,"Die Bitlänge angegeben=" + ValToStr(n_diBitLength) + ". Wert muss zwischen 1-16.","???"];
			st_MsgBoxLine4:=["Please Check Configuration.","Bitte Überprüfe Konfiguration.","???"];
			n_MsgBoxAnswer:= UIMessageBox (\Header:=st_MsgBoxHeader{n_Sp}\MsgArray:=[" "," ",st_MsgBoxLine3{n_Sp},st_MsgBoxLine4{n_Sp}," "]\Buttons:=btnOK\Icon:=iconError) ;

			STOP;
		ENDWHILE

	ELSEIF n_LastBitNr>32 THEN
		!Check last bit number

		WHILE TRUE DO
			TPErase;
			st_MsgBoxHeader:=["GetGIValue Signal="+ st_diSignalDesc ,"GetGIValue Signal="+ st_diSignalDesc,"???"];
			st_MsgBoxLine3:=["The first Bit specified=" + ValToStr(n_FirstBitNr) + " + length specified=" + ValToStr(n_diBitLength) + " is >32.","Die Erstes Bit angegeben=" + ValToStr(n_FirstBitNr) + " + Länge angegeben=" + ValToStr(n_diBitLength) + " ist >32.","???"];
			st_MsgBoxLine4:=["Please Check Configuration.","Bitte Überprüfe Konfiguration.","???"];
			n_MsgBoxAnswer:= UIMessageBox (\Header:=st_MsgBoxHeader{n_Sp}\MsgArray:=[" "," ",st_MsgBoxLine3{n_Sp},st_MsgBoxLine4{n_Sp}," "]\Buttons:=btnOK\Icon:=iconError) ;

			STOP;
		ENDWHILE

	ELSE !n_diBitLength<1
		n_ScrollNr:=0.5;
		n_ValueCount:=0;

		FOR n_CharNr FROM n_FirstBitNr	TO n_LastBitNr DO
			n_ScrollNr:=n_ScrollNr*2;

			IF n_CharNr<10 AND n_CharFirstNumber<>n_diSignal_Length THEN
				st_tempString:=st_diSignalDesc1 +"0" + ValToStr(n_CharNr) + st_diSignalDesc2;
			ELSE
				st_tempString:=st_diSignalDesc1 + ValToStr(n_CharNr) + st_diSignalDesc2;
			ENDIF

			AliasIO st_tempString, di_Temp;

			IF di_Temp = 1 THEN
				n_ValueCount:=n_ValueCount + n_ScrollNr ;
			ENDIF

		ENDFOR

		n_LastGroupInput:=n_ValueCount;
		RETURN n_ValueCount ;
	ENDIF !n_diBitLength<1
ENDIF !n_diSignal_Length

ERROR
!** Error Handler **

TEST  ERRNO
CASE ERR_ALIASIO_DEF,ERR_ALIASIO_TYPE :
	WHILE TRUE DO
		TPErase;
		st_MsgBoxHeader:=["GetGIValue Signal=" + st_tempString ,"GetGIValue Signal=" + st_tempString,"???"];
		st_MsgBoxLine3:=["Signal is missing or incorrectly defined","IO Signal ist nicht vorhanden oder Falsch geschrieben","???"];
		st_MsgBoxLine4:=["Please Check Configuration.","Bitte Überprüfe Konfiguration.","???"];
		n_MsgBoxAnswer:= UIMessageBox (\Header:=st_MsgBoxHeader{n_Sp}\MsgArray:=[" "," ",st_MsgBoxLine3{n_Sp},st_MsgBoxLine4{n_Sp}," "]\Buttons:=btnOK\Icon:=iconError) ;

		STOP;
	ENDWHILE
DEFAULT :
	WHILE TRUE DO
		TPErase;
		st_MsgBoxHeader:=["GetGIValue Unknown Error =" + ValToStr(Errno) ,"GetGIValue unbekannter Fehler =" + ValToStr(Errno),"???"];
		st_MsgBoxLine3:=["Support Required.","Unterstützung erforderlich.","???"];
		st_MsgBoxLine4:=[" "," ","???"];
		n_MsgBoxAnswer:= UIMessageBox (\Header:=st_MsgBoxHeader{n_Sp}\MsgArray:=[" "," ",st_MsgBoxLine3{n_Sp},st_MsgBoxLine4{n_Sp}," "]\Buttons:=btnOK\Icon:=iconError) ;

		STOP;
	ENDWHILE
ENDTEST

ENDFUNC !(GetGroupIP)


!*******************************************************************************


FUNC Num GetGroupIP_Bit (VAR Signaldi diSignalName,Num n_diBitLength\Switch ReturnBitOffset)
!***************************************
!* Procedure to return a numeric value *
!*    from a group of Digital Inputs   *
!* providing only one input is logic 1 *
!***************************************

VAR signaldi di_Temp;

VAR Num n_FirstBitNr;
VAR Num n_FirstBitNrMem:=0;
VAR Num n_LastBitNr;
VAR Num n_diSignal_Length;
VAR Num n_CharNr;
VAR Num n_ScrollNr;
VAR Num n_CharFirstNumber;
VAR Num n_CharLastNumber;
VAR Num n_CharNumberCount;
VAR Num n_NumberCharlength;

VAR String st_diSignalName;
VAR String st_FirstbitNr;
VAR String st_diSignalDesc;
VAR String st_diSignalDesc1;
VAR String st_diSignalDesc2;
VAR String st_tempString ;

!Stop advance pointer
WaitTime\Inpos, 0.0 ;

!Check first bit configured is a valid input
st_diSignalName:=ArgName(diSignalName);
AliasIO st_diSignalName, di_Temp;

!Check input name length
n_diSignal_Length:=StrLen(st_diSignalName);

IF n_diSignal_Length > 3 THEN
	!Determine which characters the Bit numbers start
	n_CharFirstNumber:=StrFind(st_diSignalName,1,STR_DIGIT) ;

	!Determine how many characters are numeric
	IF n_CharFirstNumber<n_diSignal_Length THEN
		n_CharLastNumber:=StrFind(st_diSignalName,n_CharFirstNumber+1,STR_DIGIT);
	ELSE
		n_CharLastNumber:=n_diSignal_Length;
	ENDIF

	n_NumberCharlength:=n_CharLastNumber-n_CharFirstNumber +1;

	!Check that there are numbers in signal description
	WHILE n_CharFirstNumber>n_diSignal_Length DO
		TPErase;
		st_MsgBoxHeader:=["GetGiBitValue  Signal=" + st_diSignalName ,"GetGiBitValue  Signal=" + st_diSignalName,"???"];
		st_MsgBoxLine3:=["There are no bit numbers in the signal name defined." ,"Es gibt keine Bit-Zahlen in der Signal-Namen definiert","???"];
		st_MsgBoxLine4:=["Please check Configuration.","Bitte Überprüfe Konfiguration.","???"];
		n_MsgBoxAnswer:= UIMessageBox (\Header:=st_MsgBoxHeader{n_Sp}\MsgArray:=[" "," ",st_MsgBoxLine3{n_Sp},st_MsgBoxLine4{n_Sp}," "]\Buttons:=btnOK\Icon:=iconError) ;

		STOP;
	ENDWHILE

	n_CharNumberCount:=1;

	!Check how many characters are numbers
	FOR n_CharNr FROM n_CharFirstNumber +1 TO n_diSignal_Length DO
		IF StrFind(st_diSignalName,n_CharNr,STR_DIGIT)<=n_diSignal_Length THEN
			INCR n_CharNumberCount ;
		ENDIF
	ENDFOR

	!Check that there are no more than 3 numbers in the signal description
	WHILE n_CharNumberCount>2 DO
		TPErase;
		st_MsgBoxHeader:=["GetGiBitValue  Signal=" + st_diSignalName ,"GetGiBitValue  Signal=" + st_diSignalName,"???"];
		st_MsgBoxLine3:=["There are more than two numbers in the" ,"Es gibt mehr als zwei Zahlen in der","???"];
		st_MsgBoxLine4:=["signal name defined. Check Configuration.","Signal-Name definiert. Konfiguration prüfen.","???"];
		n_MsgBoxAnswer:= UIMessageBox (\Header:=st_MsgBoxHeader{n_Sp}\MsgArray:=[" "," ",st_MsgBoxLine3{n_Sp},st_MsgBoxLine4{n_Sp}," "]\Buttons:=btnOK\Icon:=iconError) ;

		STOP;
	ENDWHILE

	!Check that there are no less than numbers in signal description
	WHILE n_CharNumberCount<2 DO
		TPErase;
		st_MsgBoxHeader:=["GetGiBitValue  Signal=" + st_diSignalName ,"GetGiBitValue  Signal=" + st_diSignalName,"???"];
		st_MsgBoxLine3:=["The are less than two numbers in the" ,"Das sind weniger als zwei Zahlen in der","???"];
		st_MsgBoxLine4:=["signal name defined. Check Configuration.","Signal-Name definiert. Konfiguration prüfen.","???"];
		n_MsgBoxAnswer:= UIMessageBox (\Header:=st_MsgBoxHeader{n_Sp}\MsgArray:=[" "," ",st_MsgBoxLine3{n_Sp},st_MsgBoxLine4{n_Sp}," "]\Buttons:=btnOK\Icon:=iconError) ;

		STOP;
	ENDWHILE

	!Get Bit number as a string
	st_FirstbitNr:=StrPart(st_diSignalName,n_CharFirstNumber,n_NumberCharlength);

	!Check st_FirstbitNr is a number
	WHILE StrToVal(st_FirstbitNr,n_FirstBitNr)<>TRUE DO
		TPErase;
		st_MsgBoxHeader:=["GetGiBitValue  Signal=" + st_diSignalName ,"GetGiBitValue  Signal=" + st_diSignalName ,"???"];
		st_MsgBoxLine3:=["There are not two consecutive bit numbers defined." ,"Es gibt nicht zwei aufeinander folgenden Bit-Zahlen definiert.","???"];
		st_MsgBoxLine4:=["Please Check Configuration.","Bitte Überprüfe Konfiguration.","???"];
		n_MsgBoxAnswer:= UIMessageBox (\Header:=st_MsgBoxHeader{n_Sp}\MsgArray:=[" "," ",st_MsgBoxLine3{n_Sp},st_MsgBoxLine4{n_Sp}," "]\Buttons:=btnOK\Icon:=iconError) ;

		STOP;
	ENDWHILE

	st_diSignalDesc1:=StrPart(st_diSignalName,1,n_CharFirstNumber-1);

	IF (n_CharFirstNumber+1)=n_diSignal_Length OR n_CharFirstNumber=n_diSignal_Length THEN
		!Bit numbers are the last or last two characters
		st_diSignalDesc2:="" ;
		st_diSignalDesc:=st_diSignalDesc1 + "??" ;
	ELSE
		st_diSignalDesc2:=StrPart(st_diSignalName,n_CharFirstNumber+2,n_diSignal_Length-n_CharFirstNumber-1);
		st_diSignalDesc:=st_diSignalDesc1 + "??" + st_diSignalDesc2 ;
	ENDIF

	n_LastBitNr:=n_FirstBitNr+n_diBitLength-1;

	IF n_diBitLength<1 OR n_diBitLength>16 THEN
		!Check n_diBitLength paramater is valid

		WHILE TRUE DO
			TPErase;
			st_MsgBoxHeader:=["GetGiBitValue Signal=" + st_diSignalDesc ,"GetGiBitValue Signal=" + st_diSignalDesc,"???"];
			st_MsgBoxLine3:=["The Bit length Specified=" + ValToStr(n_diBitLength) + ". Value must be between 1-16." ,"Die Bitlänge angegeben=" + ValToStr(n_diBitLength) + ". Wert muss zwischen 1-16.","???"];
			st_MsgBoxLine4:=["Please Check Configuration.","Bitte Überprüfe Konfiguration.","???"];
			n_MsgBoxAnswer:= UIMessageBox (\Header:=st_MsgBoxHeader{n_Sp}\MsgArray:=[" "," ",st_MsgBoxLine3{n_Sp},st_MsgBoxLine4{n_Sp}," "]\Buttons:=btnOK\Icon:=iconError) ;

			STOP;
		ENDWHILE

	ELSEIF n_LastBitNr>32 THEN
		!Check last bit number

		WHILE TRUE DO
			TPErase;
			st_MsgBoxHeader:=["GetGiBitValue Signal="+ st_diSignalDesc ,"GetGiBitValue Signal="+ st_diSignalDesc,"???"];
			st_MsgBoxLine3:=["The first Bit specified=" + ValToStr(n_FirstBitNr) + " + length specified=" + ValToStr(n_diBitLength) + " is >32.","Die Erstes Bit angegeben=" + ValToStr(n_FirstBitNr) + " + Länge angegeben=" + ValToStr(n_diBitLength) + " ist >32.","???"];
			st_MsgBoxLine4:=["Please Check Configuration.","Bitte Überprüfe Konfiguration.","???"];
			n_MsgBoxAnswer:= UIMessageBox (\Header:=st_MsgBoxHeader{n_Sp}\MsgArray:=[" "," ",st_MsgBoxLine3{n_Sp},st_MsgBoxLine4{n_Sp}," "]\Buttons:=btnOK\Icon:=iconError) ;

			STOP;
		ENDWHILE

	ELSE !n_diBitLength<1
		n_ScrollNr:=0;

		FOR n_CharNr FROM n_FirstBitNr	TO n_LastBitNr DO
			INCR n_ScrollNr ;

			IF n_CharNr<10 AND n_CharFirstNumber<>n_diSignal_Length THEN
				st_tempString:=st_diSignalDesc1 +"0" + ValToStr(n_CharNr) + st_diSignalDesc2;
			ELSE
				st_tempString:=st_diSignalDesc1 + ValToStr(n_CharNr) + st_diSignalDesc2;
			ENDIF

			AliasIO st_tempString, di_Temp;

			IF di_Temp = 1 THEN
				IF n_FirstBitNrMem= 0 THEN
					IF Present(ReturnBitOffset) THEN
						n_FirstBitNrMem:=n_CharNr;
					ELSE
						n_FirstBitNrMem:=n_ScrollNr;
					ENDIF
				ELSE
					RETURN 0;
				ENDIF
			ENDIF

		ENDFOR

		RETURN n_FirstBitNrMem;

	ENDIF !n_diBitLength<1
ENDIF !n_diSignal_Length

RETURN 0;

ERROR
!** Error Handler **

TEST  ERRNO
CASE ERR_ALIASIO_DEF,ERR_ALIASIO_TYPE :
	WHILE TRUE DO
		TPErase;
		st_MsgBoxHeader:=["GetGiBitValue Signal=" + st_tempString ,"GetGiBitValue Signal=" + st_tempString,"???"];
		st_MsgBoxLine3:=["Signal is missing or incorrectly defined","IO Signal ist nicht vorhanden oder Falsch geschrieben","???"];
		st_MsgBoxLine4:=["Please Check Configuration.","Bitte Überprüfe Konfiguration.","???"];
		n_MsgBoxAnswer:= UIMessageBox (\Header:=st_MsgBoxHeader{n_Sp}\MsgArray:=[" "," ",st_MsgBoxLine3{n_Sp},st_MsgBoxLine4{n_Sp}," "]\Buttons:=btnOK\Icon:=iconError) ;

		STOP;
	ENDWHILE
DEFAULT :
	WHILE TRUE DO
		TPErase;
		st_MsgBoxHeader:=["GetGiBitValue Unknown Error =" + ValToStr(Errno) ,"GetGiBitValue unbekannter Fehler =" + ValToStr(Errno),"???"];
		st_MsgBoxLine3:=["Support Required.","Unterstützung erforderlich.","???"];
		st_MsgBoxLine4:=[" "," ","???"];
		n_MsgBoxAnswer:= UIMessageBox (\Header:=st_MsgBoxHeader{n_Sp}\MsgArray:=[" "," ",st_MsgBoxLine3{n_Sp},st_MsgBoxLine4{n_Sp}," "]\Buttons:=btnOK\Icon:=iconError) ;

		STOP;
	ENDWHILE
ENDTEST

ENDFUNC !(GetGroupIP_Bit)


!*******************************************************************************


FUNC Num GetGroupOP (VAR Signaldo doSignalName,Num n_doBitLength)
!***************************************
!* Procedure to return a numeric value *
!*   from a group of Digital Outputs   *
!***************************************

VAR signaldo do_Temp;

VAR Num n_FirstBitNr;
VAR Num n_LastBitNr;
VAR Num n_doSignal_Length;
VAR Num n_CharNr;
VAR Num n_ScrollNr;
VAR Num n_ValueCount;
VAR Num n_CharFirstNumber;
VAR Num n_CharLastNumber;
VAR Num n_CharNumberCount;
VAR Num n_NumberCharlength;

VAR String st_doSignalName;
VAR String st_FirstbitNr;
VAR String st_doSignalDesc;
VAR String st_doSignalDesc1;
VAR String st_doSignalDesc2;
VAR String st_tempString ;

!Stop advance pointer
WaitTime\Inpos, 0.0 ;

!Check first bit configured is a valid output
st_doSignalName:=ArgName(doSignalName);
AliasIO st_doSignalName, do_Temp;

!Check output name length
n_doSignal_Length:=StrLen(st_doSignalName);

IF n_doSignal_Length > 3 THEN
	!Determine which characters the Bit numbers start
	n_CharFirstNumber:=StrFind(st_doSignalName,1,STR_DIGIT) ;

	!Determine how many characters are numeric
	IF n_CharFirstNumber<n_doSignal_Length THEN
		n_CharLastNumber:=StrFind(st_doSignalName,n_CharFirstNumber+1,STR_DIGIT);
	ELSE
		n_CharLastNumber:=n_doSignal_Length;
	ENDIF

	n_NumberCharlength:=n_CharLastNumber-n_CharFirstNumber +1;

	!Check that there are numbers in signal description
	WHILE n_CharFirstNumber>n_doSignal_Length DO
		TPErase;
		st_MsgBoxHeader:=["GetGOValue  Signal=" + st_doSignalName ,"GetGOValue  Signal=" + st_doSignalName,"???"];
		st_MsgBoxLine3:=["There are no bit numbers in the signal name defined." ,"Es gibt keine Bit-Zahlen in der Signal-Namen definiert","???"];
		st_MsgBoxLine4:=["Check Configuration","Überprüfe Konfiguration","???"];
		n_MsgBoxAnswer:= UIMessageBox (\Header:=st_MsgBoxHeader{n_Sp}\MsgArray:=[" "," ",st_MsgBoxLine3{n_Sp},st_MsgBoxLine4{n_Sp}," "]\Buttons:=btnOK\Icon:=iconError) ;

		STOP;
	ENDWHILE

	n_CharNumberCount:=1;

	!Check how many characters are numbers
	FOR n_CharNr FROM n_CharFirstNumber +1 TO n_doSignal_Length DO
		IF StrFind(st_doSignalName,n_CharNr,STR_DIGIT)<=n_doSignal_Length THEN
			INCR n_CharNumberCount ;
		ENDIF
	ENDFOR

